// TIA Portal project "TM20T_TiaV151_S71200_V17" (V17)

(* hardware
DEVICE "S7-1200 station_1"  S7-1200 Station
   slot 0: "Rack_0"  S7-1200 Rack  Rack  V1.0
   slot 1: "PLC_1"  CPU 1214C DC/DC/DC  6ES7 214-1AG40-0XB0  V4.2
   slot 2: "DI 8x24VDC_1"  6ES7 221-1BF32-0XB0  V2.0
   slot 3: "DI 16x24VDC_1"  SM 1221 DI16 x 24VDC  6ES7 221-1BH30-0XB0  V1.0
   slot 4: "DI 16x24VDC_2"  SM 1221 DI16 x 24VDC  6ES7 221-1BH30-0XB0  V1.0
   slot 5: "DI 16x24VDC_3"  SM 1221 DI16 x 24VDC  6ES7 221-1BH30-0XB0  V1.0
DEVICE "PC-System_1"  SIMATIC PC station
   slot 0: "SIMATIC PC station"  Rail  SIMATIC PC-Station  V1.0
      slot 125: "Stationmanager"  Station_Manager  V6.0.4
   slot 1: "HMI_RT_1"  WinCC RT Advanced  6AV2 104-0xxxx-xxxx  17.0.0.0
      slot 33792: "Computer interface"  Host interface
   slot 2: "IE general_1"  IE General  IE_CP  V8.2.0
*)

// ===== PLC "PLC_1"  CPU 1214C DC/DC/DC =====

VAR_GLOBAL   // PLC tag table "Default tag table"
   "System_Byte" AT %MB1 : Byte;
   "FirstScan" AT %M1.0 : Bool;
   "DiagStatusUpdate" AT %M1.1 : Bool;
   "AlwaysTRUE" AT %M1.2 : Bool;
   "AlwaysFALSE" AT %M1.3 : Bool;
   "Clock_Byte" AT %MB0 : Byte;
   "Clock_10Hz" AT %M0.0 : Bool;
   "Clock_5Hz" AT %M0.1 : Bool;
   "Clock_2.5Hz" AT %M0.2 : Bool;
   "Clock_2Hz" AT %M0.3 : Bool;
   "Clock_1.25Hz" AT %M0.4 : Bool;
   "Clock_1Hz" AT %M0.5 : Bool;
   "Clock_0.625Hz" AT %M0.6 : Bool;
   "Clock_0.5Hz" AT %M0.7 : Bool;
END_VAR

VAR_GLOBAL   // PLC tag table "INPUT"
   "I_F1_Up" AT %I0.0 : Bool;   // Tầng 1 gọi đi lên
   "I_F2_Up" AT %I0.1 : Bool;   // Tầng 2 gọi đi lên
   "I_F3_Up" AT %I0.2 : Bool;   // Tầng 3 gọi đi lên
   "I_F2_Down" AT %I0.3 : Bool;   // Tầng 2 gọi đi xuống
   "I_F3_Down" AT %I0.4 : Bool;   // Tầng 3 gọi đi xuống
   "I_F4_Down" AT %I0.5 : Bool;   // Tầng 4 gọi đi xuống
   "I_Inside_F1" AT %I0.6 : Bool;   // Gọi tầng trong thang máy gọi tầng 1
   "I_Inside_F2" AT %I0.7 : Bool;   // Gọi tầng trong thang máy gọi tầng 2
   "I_Inside_F3" AT %I1.0 : Bool;   // Gọi tầng trong thang máy gọi tầng 3
   "I_Inside_F4" AT %I1.1 : Bool;   // Gọi tầng trong thang máy gọi tầng 4
   "I_Inside_Door_Open" AT %I1.2 : Bool;   // Nút nhấn mở cửa trong thang máy
   "I_Inside_Door_Close" AT %I1.3 : Bool;   // Nút nhấn đóng cửa trong thang máy
   "I_Cabin_Position" AT %I1.4 : Bool;   // Cảm biến vị trí buồng thang
   "I_Door_Opened" AT %I1.5 : Bool;   // Limits Switch cữa đã mở
   "I_Door_Closed" AT %I1.6 : Bool;   // Limit Switch cửa đã đóng
   "I_F4_Up" AT %I1.7 : Bool;
   "I_F5_Up" AT %I2.0 : Bool;
   "I_F6_Up" AT %I2.1 : Bool;
   "I_F7_Up" AT %I2.2 : Bool;
   "I_F8_Up" AT %I2.3 : Bool;
   "I_F9_Up" AT %I2.4 : Bool;
   "I_F10_Up" AT %I2.5 : Bool;
   "I_F11_Up" AT %I2.6 : Bool;
   "I_F12_Up" AT %I2.7 : Bool;
   "I_F13_Up" AT %I3.0 : Bool;
   "I_F14_Up" AT %I3.1 : Bool;
   "I_F15_Up" AT %I3.2 : Bool;
   "I_F16_Up" AT %I3.3 : Bool;
   "I_F17_Up" AT %I3.4 : Bool;
   "I_F18_Up" AT %I3.5 : Bool;
   "I_F19_Up" AT %I3.6 : Bool;
   "I_F5_Down" AT %I3.7 : Bool;
   "I_F6_Down" AT %I4.0 : Bool;
   "I_F7_Down" AT %I4.1 : Bool;
   "I_F8_Down" AT %I4.2 : Bool;
   "I_F9_Down" AT %I4.3 : Bool;
   "I_F10_Down" AT %I4.4 : Bool;
   "I_F11_Down" AT %I4.5 : Bool;
   "I_F12_Down" AT %I4.6 : Bool;
   "I_F13_Down" AT %I4.7 : Bool;
   "I_F14_Down" AT %I5.0 : Bool;
   "I_F15_Down" AT %I5.1 : Bool;
   "I_F16_Down" AT %I5.2 : Bool;
   "I_F17_Down" AT %I5.3 : Bool;
   "I_F18_Down" AT %I5.4 : Bool;
   "I_F19_Down" AT %I5.5 : Bool;
   "I_F20_Down" AT %I5.6 : Bool;
   "I_Inside_F1(1)" AT %I5.7 : Bool;
   "I_Inside_F2(1)" AT %I6.0 : Bool;
   "I_Inside_F3(1)" AT %I6.1 : Bool;
   "I_Inside_F4(1)" AT %I6.2 : Bool;
   "I_Inside_F5" AT %I6.3 : Bool;
   "I_Inside_F6" AT %I6.4 : Bool;
   "I_Inside_F7" AT %I6.5 : Bool;
   "I_Inside_F8" AT %I6.6 : Bool;
   "I_Inside_F9" AT %I6.7 : Bool;
   "I_Inside_F10" AT %I7.0 : Bool;
   "I_Inside_F11" AT %I7.1 : Bool;
   "I_Inside_F12" AT %I7.2 : Bool;
   "I_Inside_F13" AT %I7.3 : Bool;
   "I_Inside_F14" AT %I7.4 : Bool;
   "I_Inside_F15" AT %I7.5 : Bool;
   "I_Inside_F16" AT %I7.6 : Bool;
   "I_Inside_F17" AT %I7.7 : Bool;
   "I_Inside_F18" AT %I8.0 : Bool;
   "I_Inside_F19" AT %I8.1 : Bool;
   "I_Inside_F20" AT %I8.2 : Bool;
END_VAR

VAR_GLOBAL   // PLC tag table "OUTPUT"
   "Q_Door_Open" AT %Q0.0 : Bool;   // Cửa buồng thang mở
   "Q_Door_Close" AT %Q0.1 : Bool;   // Cửa buồng thang đóng
   "Q_Eleveytor_Up" AT %Q0.2 : Bool;   // Thang máy đi lên
   "Q_Eleveytor_Down" AT %Q0.3 : Bool;   // Thang máy đi xuống
END_VAR

VAR_GLOBAL   // PLC tag table "xung suon len"
   "P1" AT %M20.0 : Bool;
   "P2" AT %M20.1 : Bool;
   "P3" AT %M20.2 : Bool;
   "P4" AT %M20.3 : Bool;
   "P5" AT %M20.4 : Bool;
   "P6" AT %M20.5 : Bool;
   "P7" AT %M20.6 : Bool;
   "P8" AT %M20.7 : Bool;
   "P9" AT %M21.0 : Bool;
   "P10" AT %M21.1 : Bool;
   "P11" AT %M21.2 : Bool;
   "P12" AT %M21.3 : Bool;
   "P13" AT %M21.4 : Bool;
   "P14" AT %M21.5 : Bool;
   "P15" AT %M21.6 : Bool;
   "P16" AT %M21.7 : Bool;
   "P17" AT %M22.0 : Bool;
   "P18" AT %M22.1 : Bool;
   "P19" AT %M22.2 : Bool;
   "P20" AT %M22.3 : Bool;
   "P21" AT %M22.4 : Bool;
   "P22" AT %M22.5 : Bool;
   "P23" AT %M22.6 : Bool;
   "P24" AT %M22.7 : Bool;
   "P25" AT %M23.0 : Bool;
   "P26" AT %M23.1 : Bool;
   "P27" AT %M23.2 : Bool;
   "P28" AT %M23.3 : Bool;
   "P29" AT %M23.4 : Bool;
   "P30" AT %M23.5 : Bool;
   "P31" AT %M23.6 : Bool;
   "P32" AT %M23.7 : Bool;
   "P33" AT %M24.0 : Bool;
   "P34" AT %M24.1 : Bool;
   "P35" AT %M24.2 : Bool;
   "P36" AT %M24.3 : Bool;
   "P37" AT %M24.4 : Bool;
   "P38" AT %M24.5 : Bool;
   "P39" AT %M24.6 : Bool;
   "P40" AT %M24.7 : Bool;
   "P41" AT %M25.0 : Bool;
   "P42" AT %M25.1 : Bool;
   "P43" AT %M25.2 : Bool;
   "P44" AT %M25.3 : Bool;
   "P45" AT %M25.4 : Bool;
   "P46" AT %M25.5 : Bool;
   "P47" AT %M25.6 : Bool;
   "P48" AT %M25.7 : Bool;
   "P49" AT %M26.0 : Bool;
   "P50" AT %M26.1 : Bool;
   "P51" AT %M26.2 : Bool;
   "P52" AT %M26.3 : Bool;
   "P53" AT %M26.4 : Bool;
   "P54" AT %M26.5 : Bool;
   "P55" AT %M26.6 : Bool;
   "P56" AT %M26.7 : Bool;
   "P57" AT %M27.0 : Bool;
   "P58" AT %M27.1 : Bool;
   "P59" AT %M27.2 : Bool;
   "P60" AT %M27.3 : Bool;
   "P61" AT %M27.4 : Bool;
   "P62" AT %M27.5 : Bool;
   "P63" AT %M27.6 : Bool;
   "P64" AT %M27.7 : Bool;
   "P65" AT %M28.0 : Bool;
   "P66" AT %M28.1 : Bool;
   "P67" AT %M28.2 : Bool;
   "P68" AT %M28.3 : Bool;
   "P69" AT %M28.4 : Bool;
   "P70" AT %M28.5 : Bool;
   "P71" AT %M28.6 : Bool;
   "P72" AT %M28.7 : Bool;
   "P73" AT %M29.0 : Bool;
   "P74" AT %M29.1 : Bool;
   "P75" AT %M29.2 : Bool;
   "P76" AT %M29.3 : Bool;
   "P77" AT %M29.4 : Bool;
   "P78" AT %M29.5 : Bool;
   "P79" AT %M29.6 : Bool;
   "P80" AT %M29.7 : Bool;
   "P81" AT %M30.0 : Bool;
   "P82" AT %M30.1 : Bool;
   "P83" AT %M30.2 : Bool;
   "P84" AT %M30.3 : Bool;
   "P85" AT %M30.4 : Bool;
   "P86" AT %M30.5 : Bool;
   "P87" AT %M30.6 : Bool;
   "P88" AT %M30.7 : Bool;
   "P89" AT %M31.0 : Bool;
   "P90" AT %M31.1 : Bool;
   "P91" AT %M31.2 : Bool;
   "P92" AT %M31.3 : Bool;
   "P93" AT %M31.4 : Bool;
   "P94" AT %M31.5 : Bool;
   "P95" AT %M31.6 : Bool;
   "P96" AT %M31.7 : Bool;
   "P97" AT %M32.0 : Bool;
   "P98" AT %M32.1 : Bool;
   "P99" AT %M32.2 : Bool;
   "P100" AT %M32.3 : Bool;
   "P101" AT %M32.4 : Bool;
   "P102" AT %M32.5 : Bool;
   "P103" AT %M32.6 : Bool;
   "P104" AT %M32.7 : Bool;
   "P105" AT %M33.0 : Bool;
   "P106" AT %M33.1 : Bool;
   "P107" AT %M33.2 : Bool;
   "P108" AT %M33.3 : Bool;
   "P109" AT %M33.4 : Bool;
   "P110" AT %M33.5 : Bool;
   "P111" AT %M33.6 : Bool;
   "P112" AT %M33.7 : Bool;
   "P113" AT %M34.0 : Bool;
   "P114" AT %M34.1 : Bool;
   "P115" AT %M34.2 : Bool;
   "P116" AT %M34.3 : Bool;
   "P117" AT %M34.4 : Bool;
   "P118" AT %M34.5 : Bool;
   "P119" AT %M34.6 : Bool;
   "P120" AT %M34.7 : Bool;
   "P121" AT %M35.0 : Bool;
   "P122" AT %M35.1 : Bool;
   "P123" AT %M35.2 : Bool;
   "P124" AT %M35.3 : Bool;
   "P125" AT %M35.4 : Bool;
   "P126" AT %M35.5 : Bool;
   "P127" AT %M35.6 : Bool;
   "P128" AT %M35.7 : Bool;
   "P129" AT %M36.0 : Bool;
   "P130" AT %M36.1 : Bool;
   "P131" AT %M36.2 : Bool;
   "P132" AT %M36.3 : Bool;
   "P133" AT %M36.4 : Bool;
   "P134" AT %M36.5 : Bool;
   "P135" AT %M36.6 : Bool;
   "P136" AT %M36.7 : Bool;
   "P137" AT %M37.0 : Bool;
   "P138" AT %M37.1 : Bool;
   "P139" AT %M37.2 : Bool;
   "P140" AT %M37.3 : Bool;
   "P141" AT %M37.4 : Bool;
   "P142" AT %M37.5 : Bool;
   "P143" AT %M37.6 : Bool;
   "P144" AT %M37.7 : Bool;
   "P145" AT %M38.0 : Bool;
   "P146" AT %M38.1 : Bool;
   "P147" AT %M38.2 : Bool;
   "P148" AT %M38.3 : Bool;
   "P149" AT %M38.4 : Bool;
   "P150" AT %M38.5 : Bool;
   "P151" AT %M38.6 : Bool;
   "P152" AT %M38.7 : Bool;
   "P153" AT %M39.0 : Bool;
   "P154" AT %M39.1 : Bool;
   "P155" AT %M39.2 : Bool;
   "P156" AT %M39.3 : Bool;
   "P157" AT %M39.4 : Bool;
   "P158" AT %M39.5 : Bool;
   "P159" AT %M39.6 : Bool;
   "P160" AT %M39.7 : Bool;
   "P161" AT %M40.0 : Bool;
   "P162" AT %M40.1 : Bool;
   "P163" AT %M40.2 : Bool;
   "P164" AT %M40.3 : Bool;
   "P165" AT %M40.4 : Bool;
   "P166" AT %M40.5 : Bool;
   "P167" AT %M40.6 : Bool;
   "P168" AT %M40.7 : Bool;
   "P169" AT %M41.0 : Bool;
   "P170" AT %M41.1 : Bool;
   "P171" AT %M41.2 : Bool;
   "P172" AT %M41.3 : Bool;
   "P173" AT %M41.4 : Bool;
   "P174" AT %M41.5 : Bool;
   "P175" AT %M41.6 : Bool;
   "P176" AT %M41.7 : Bool;
   "P177" AT %M42.0 : Bool;
   "P178" AT %M42.1 : Bool;
   "P179" AT %M42.2 : Bool;
   "P180" AT %M42.3 : Bool;
   "P181" AT %M42.4 : Bool;
   "P182" AT %M42.5 : Bool;
   "P183" AT %M42.6 : Bool;
   "P184" AT %M42.7 : Bool;
   "P185" AT %M43.0 : Bool;
   "P186" AT %M43.1 : Bool;
   "P187" AT %M43.2 : Bool;
   "P188" AT %M43.3 : Bool;
   "P189" AT %M43.4 : Bool;
   "P190" AT %M43.5 : Bool;
   "P191" AT %M43.6 : Bool;
   "P192" AT %M43.7 : Bool;
   "P193" AT %M44.0 : Bool;
   "P194" AT %M44.1 : Bool;
   "P195" AT %M44.2 : Bool;
   "P196" AT %M44.3 : Bool;
   "P197" AT %M44.4 : Bool;
   "P198" AT %M44.5 : Bool;
   "P199" AT %M44.6 : Bool;
   "P200" AT %M44.7 : Bool;
   "P201" AT %M45.0 : Bool;
   "P202" AT %M45.1 : Bool;
   "P203" AT %M45.2 : Bool;
   "P204" AT %M45.3 : Bool;
   "P205" AT %M45.4 : Bool;
   "P206" AT %M45.5 : Bool;
   "P207" AT %M45.6 : Bool;
   "P208" AT %M45.7 : Bool;
   "P209" AT %M46.0 : Bool;
   "P210" AT %M46.1 : Bool;
   "P211" AT %M46.2 : Bool;
   "P212" AT %M46.3 : Bool;
   "P213" AT %M46.4 : Bool;
   "P214" AT %M46.5 : Bool;
   "P215" AT %M46.6 : Bool;
   "P216" AT %M46.7 : Bool;
   "P217" AT %M47.0 : Bool;
   "P218" AT %M47.1 : Bool;
   "P219" AT %M47.2 : Bool;
END_VAR

VAR_GLOBAL   // PLC tag table "Simulation"
   "Simu_Eleveytor" AT %MW100 : Int;
   "Simu_Door_F1" AT %MW102 : Int;
   "Simu_Door_F2" AT %MW104 : Int;
   "Simu_Door_F3" AT %MW106 : Int;
   "Simu_Door_F4" AT %MW108 : Int;
   "M_Simulation" AT %M10.0 : Bool;
   "Display_Inside_F2" AT %M10.1 : Bool;   // Hiển thị màu nút nhấn trong buồng thang tầng 2
   "Display_Inside_F3" AT %M10.2 : Bool;   // Hiển thị màu nút nhấn trong buồng thang tầng 3
   "Simu_Door_F5" AT %MW110 : Int;
   "Simu_Door_F6" AT %MW112 : Int;
   "Simu_Door_F7" AT %MW114 : Int;
   "Simu_Door_F8" AT %MW116 : Int;
   "Simu_Door_F9" AT %MW118 : Int;
   "Simu_Door_F10" AT %MW120 : Int;
   "Simu_Door_F11" AT %MW122 : Int;
   "Simu_Door_F12" AT %MW124 : Int;
   "Simu_Door_F13" AT %MW126 : Int;
   "Simu_Door_F14" AT %MW128 : Int;
   "Simu_Door_F15" AT %MW130 : Int;
   "Simu_Door_F16" AT %MW132 : Int;
   "Simu_Door_F17" AT %MW134 : Int;
   "Simu_Door_F18" AT %MW136 : Int;
   "Simu_Door_F19" AT %MW138 : Int;
   "Simu_Door_F20" AT %MW140 : Int;
   "Display_Inside_F4" AT %M10.3 : Bool;
   "Display_Inside_F5" AT %M10.4 : Bool;
   "Display_Inside_F6" AT %M10.5 : Bool;
   "Display_Inside_F7" AT %M10.6 : Bool;
   "Display_Inside_F8" AT %M10.7 : Bool;
   "Display_Inside_F9" AT %M11.0 : Bool;
   "Display_Inside_F10" AT %M11.1 : Bool;
   "Display_Inside_F11" AT %M11.2 : Bool;
   "Display_Inside_F12" AT %M11.3 : Bool;
   "Display_Inside_F13" AT %M11.4 : Bool;
   "Display_Inside_F14" AT %M11.5 : Bool;
   "Display_Inside_F15" AT %M11.6 : Bool;
   "Display_Inside_F16" AT %M11.7 : Bool;
   "Display_Inside_F17" AT %M12.0 : Bool;
   "Display_Inside_F18" AT %M12.1 : Bool;
   "Display_Inside_F19" AT %M12.2 : Bool;
   "M_Check1" AT %M12.3 : Bool;
   "M_Check2" AT %M12.4 : Bool;
END_VAR

TYPE "Thang_May"
   STRUCT
      Position : Bool;   // Vị trí thang máy ở tầng hiện tại
      Btt_Up_Selected : Bool;   // Đã chọn đi lên
      Btt_Down_Selected : Bool;   // Đã chọn đi xuống
      TG_Up_Selected : Bool;   // Lựa chọn đi lên đã chọn
      TG_Down_Selected : Bool;   // Lựa chọn đi xuống đã chọn
      Sensor_Correct_Position : Bool;   // Vị trí chính xác để mở cửa
      Door_Opened : Bool;   // Cửa đã mở
      Door_Closed : Bool;   // Cửa đã đóng
      I_Button_Up : Bool;   // Nút nhấn đi lên
      I_Button_Down : Bool;   // Nút nhấn đi xuống
   END_STRUCT;
END_TYPE

DATA_BLOCK "DB_Data"   // DB1
{ S7_Optimized_Access := 'TRUE' }
VERSION : 0.1
   VAR
      F1 : "Thang_May";
      F2 : "Thang_May";
      F3 : "Thang_May";
      F4 : "Thang_May";
      F20 : "Thang_May";
      F19 : "Thang_May";
      F18 : "Thang_May";
      F17 : "Thang_May";
      F16 : "Thang_May";
      F15 : "Thang_May";
      F14 : "Thang_May";
      F13 : "Thang_May";
      F12 : "Thang_May";
      F11 : "Thang_May";
      F10 : "Thang_May";
      F9 : "Thang_May";
      F8 : "Thang_May";
      F7 : "Thang_May";
      F6 : "Thang_May";
      F5 : "Thang_May";
      Button_Inside_F1 : Bool;
      Button_Inside_F2 : Bool;
      Button_Inside_F3 : Bool;
      Button_Inside_F20 : Bool;
      Button_Inside_F19 : Bool;
      Button_Inside_F18 : Bool;
      Button_Inside_F17 : Bool;
      Button_Inside_F16 : Bool;
      Button_Inside_F15 : Bool;
      Button_Inside_F14 : Bool;
      Button_Inside_F13 : Bool;
      Button_Inside_F12 : Bool;
      Button_Inside_F11 : Bool;
      Button_Inside_F10 : Bool;
      Button_Inside_F9 : Bool;
      Button_Inside_F8 : Bool;
      Button_Inside_F7 : Bool;
      Button_Inside_F6 : Bool;
      Button_Inside_F5 : Bool;
      Button_Inside_F4 : Bool;
      Button_Inside_Open : Bool;
      Button_Inside_Close : Bool;
      LS_Door_Opened : Bool;
      LS_Door_Closed : Bool;
      Eleveytor_Upping : Bool;
      Eleveytor_Downing : Bool;
      Last_Is_Up : Bool;   // Trước đó thang máy đang đi lên
      Last_Is_Down : Bool;   // Trước đó thang máy đang đi xuống
   END_VAR
BEGIN
END_DATA_BLOCK

// folder: System blocks/Program resources

DATA_BLOCK "IEC_Timer_0_DB"   // DB2
{ S7_Optimized_Access := 'TRUE' }
AUTHOR : Simatic
FAMILY : IEC
NAME : IEC_TMR
VERSION : 1.0
// stored: InstanceOfName IEC_TIMER
"IEC_TIMER"
BEGIN
END_DATA_BLOCK

DATA_BLOCK "IEC_Timer_0_DB_1"   // DB3
{ S7_Optimized_Access := 'TRUE' }
AUTHOR : Simatic
FAMILY : IEC
NAME : IEC_TMR
VERSION : 1.0
// stored: InstanceOfName IEC_TIMER
"IEC_TIMER"
BEGIN
END_DATA_BLOCK

DATA_BLOCK "IEC_Timer_0_DB_2"   // DB4
{ S7_Optimized_Access := 'TRUE' }
AUTHOR : Simatic
FAMILY : IEC
NAME : IEC_TMR
VERSION : 1.0
// stored: InstanceOfName IEC_TIMER
"IEC_TIMER"
BEGIN
END_DATA_BLOCK

DATA_BLOCK "IEC_Timer_0_DB_3"   // DB5
{ S7_Optimized_Access := 'TRUE' }
AUTHOR : Simatic
FAMILY : IEC
NAME : IEC_TMR
VERSION : 1.0
// stored: InstanceOfName IEC_TIMER
"IEC_TIMER"
BEGIN
END_DATA_BLOCK

DATA_BLOCK "IEC_Timer_0_DB_4"   // DB6
{ S7_Optimized_Access := 'TRUE' }
AUTHOR : Simatic
FAMILY : IEC
NAME : IEC_TMR
VERSION : 1.0
// stored: InstanceOfName IEC_TIMER
"IEC_TIMER"
BEGIN
END_DATA_BLOCK

// folder: (top level)

FUNCTION "FC_Nut_Nhan" : Void   // FC1, LAD
{ S7_Optimized_Access := 'TRUE' }
VERSION : 0.1
   VAR_TEMP   // added for the SCL form of the ladder/FBD networks
      _w1 : Bool;
      _w2 : Bool;
      _w3 : Bool;
      _w4 : Bool;
      _w5 : Bool;
      _w6 : Bool;
      _w7 : Bool;
      _w8 : Bool;
      _w9 : Bool;
      _w10 : Bool;
      _w11 : Bool;
      _w12 : Bool;
      _w13 : Bool;
      _w14 : Bool;
      _w15 : Bool;
      _w16 : Bool;
      _w17 : Bool;
      _w18 : Bool;
      _w19 : Bool;
      _w20 : Bool;
      _w21 : Bool;
      _w22 : Bool;
      _w23 : Bool;
      _w24 : Bool;
      _w25 : Bool;
      _w26 : Bool;
      _w27 : Bool;
   END_VAR
BEGIN

REGION Network 1: Nút nhấn MỞ cửa tại các tầng
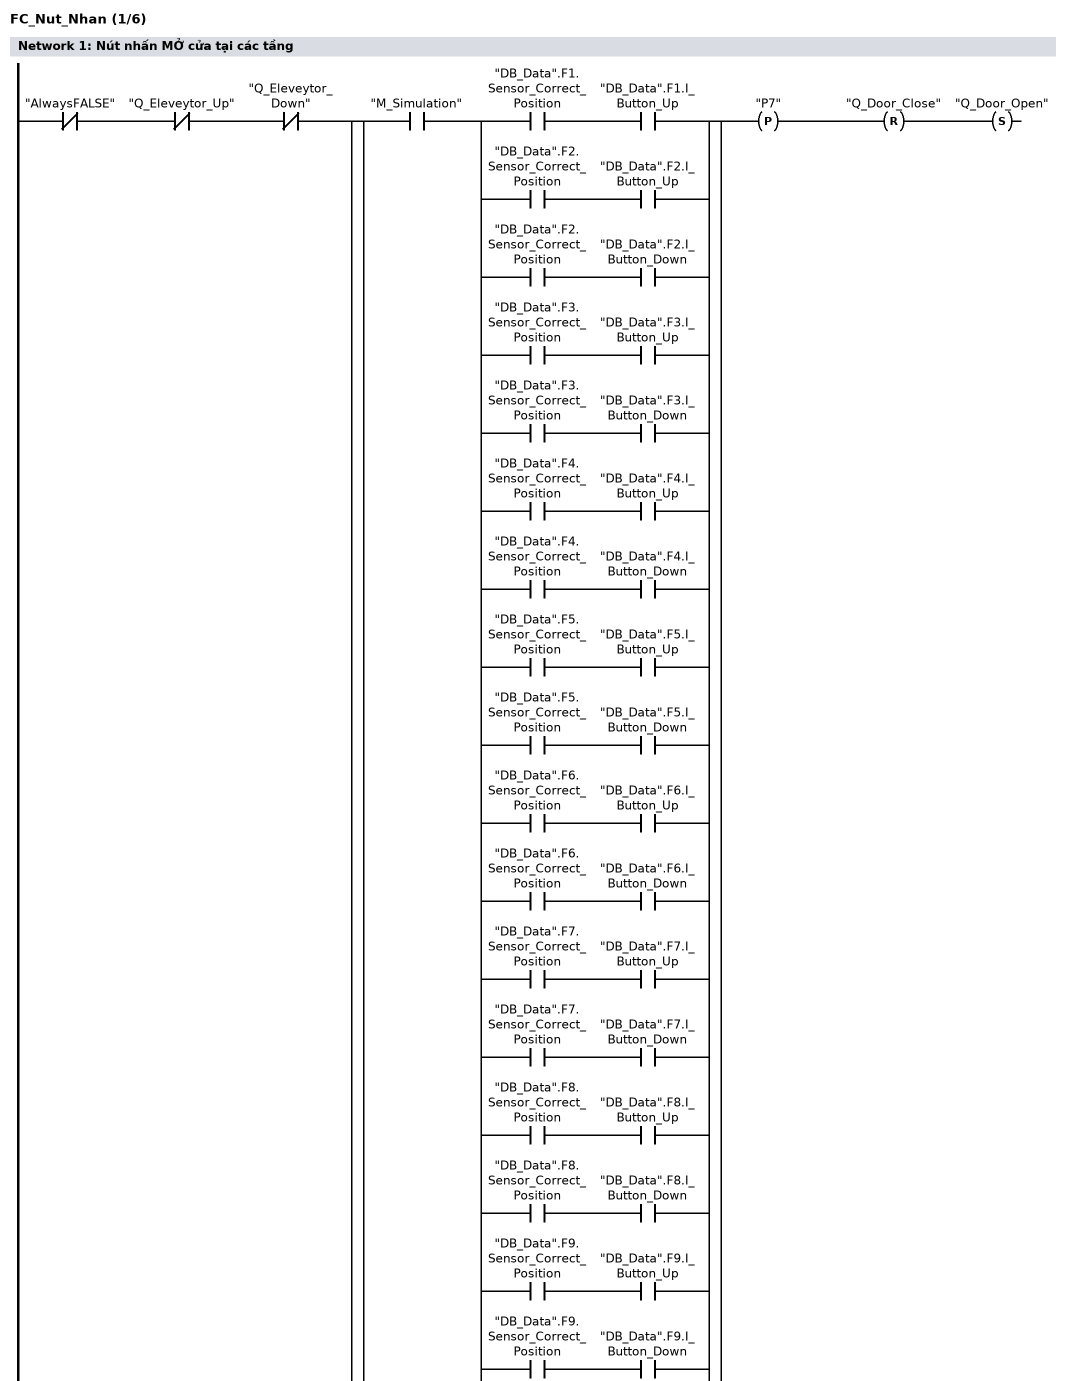
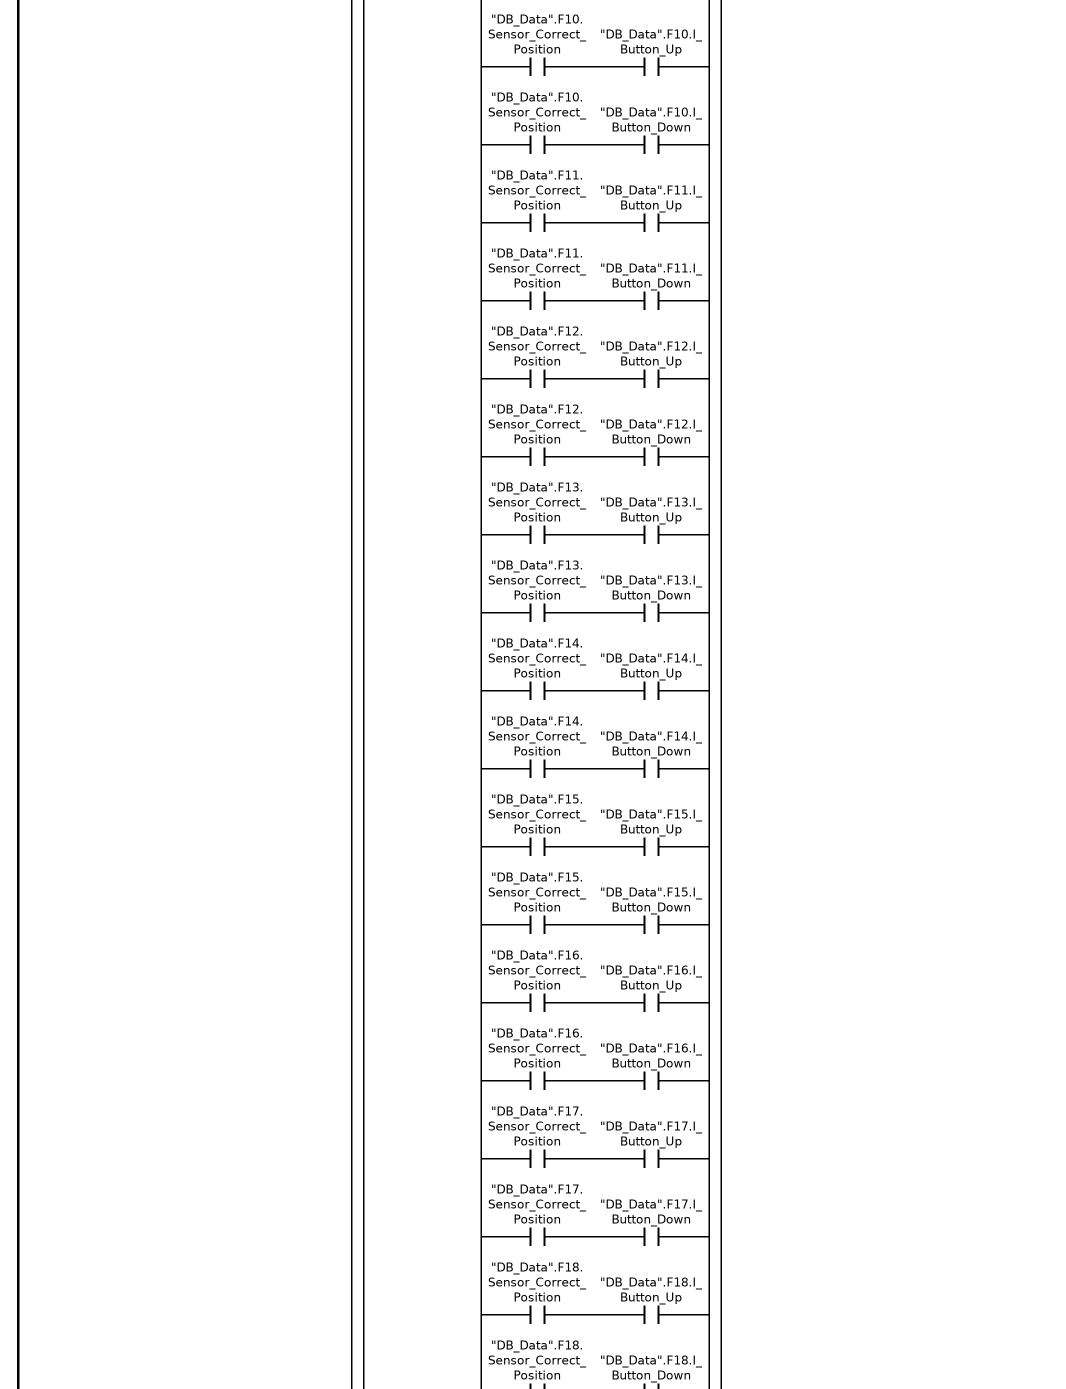
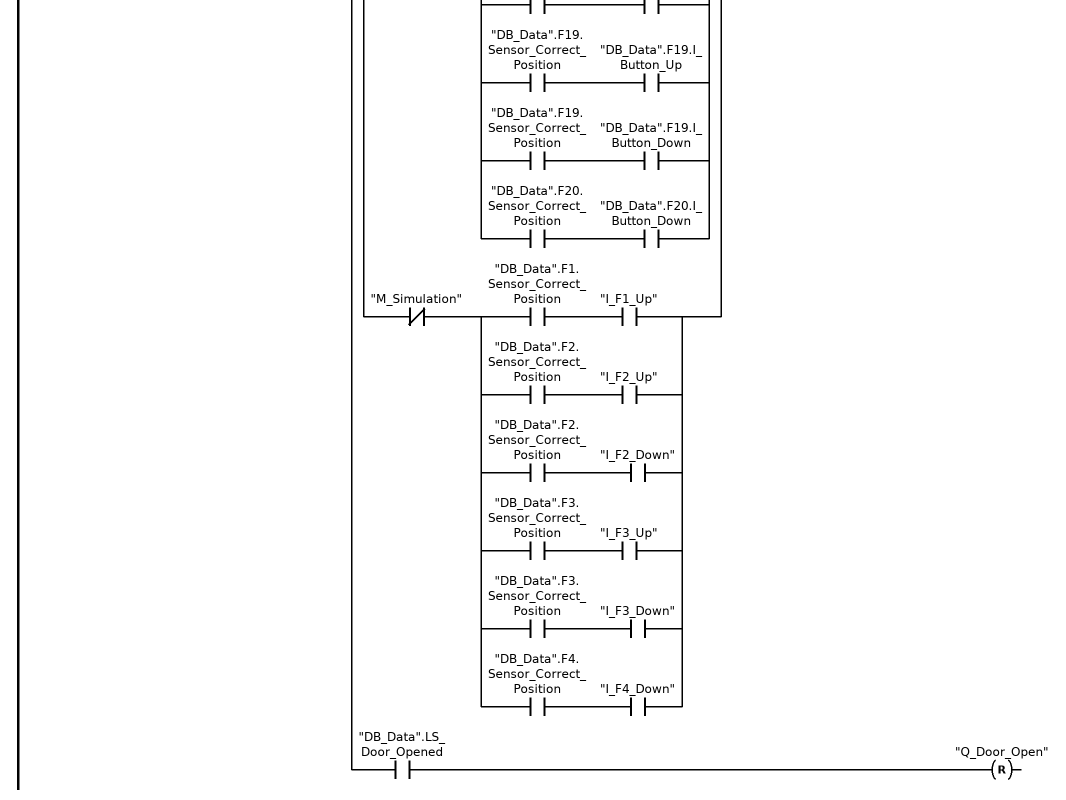
   RUNG wire#powerrail
      I_Contact( "AlwaysFALSE" )
      I_Contact( "Q_Eleveytor_Up" )
      I_Contact( "Q_Eleveytor_Down" )
      wire#w1
      Contact( "M_Simulation" )
      wire#w2
      Contact( "DB_Data".F1.Sensor_Correct_Position )
      Contact( "DB_Data".F1.I_Button_Up )
      wire#w3
      P_Trig( "P7" )
      R_Coil( "Q_Door_Close" )
      S_Coil( "Q_Door_Open" )
   END_RUNG
   RUNG wire#w2
      Contact( "DB_Data".F2.Sensor_Correct_Position )
      Contact( "DB_Data".F2.I_Button_Up )
   END_RUNG wire#w3
   RUNG wire#w2
      Contact( "DB_Data".F2.Sensor_Correct_Position )
      Contact( "DB_Data".F2.I_Button_Down )
   END_RUNG wire#w3
   RUNG wire#w2
      Contact( "DB_Data".F3.Sensor_Correct_Position )
      Contact( "DB_Data".F3.I_Button_Up )
   END_RUNG wire#w3
   RUNG wire#w2
      Contact( "DB_Data".F3.Sensor_Correct_Position )
      Contact( "DB_Data".F3.I_Button_Down )
   END_RUNG wire#w3
   RUNG wire#w2
      Contact( "DB_Data".F4.Sensor_Correct_Position )
      Contact( "DB_Data".F4.I_Button_Up )
   END_RUNG wire#w3
   RUNG wire#w2
      Contact( "DB_Data".F4.Sensor_Correct_Position )
      Contact( "DB_Data".F4.I_Button_Down )
   END_RUNG wire#w3
   RUNG wire#w2
      Contact( "DB_Data".F5.Sensor_Correct_Position )
      Contact( "DB_Data".F5.I_Button_Up )
   END_RUNG wire#w3
   RUNG wire#w2
      Contact( "DB_Data".F5.Sensor_Correct_Position )
      Contact( "DB_Data".F5.I_Button_Down )
   END_RUNG wire#w3
   RUNG wire#w2
      Contact( "DB_Data".F6.Sensor_Correct_Position )
      Contact( "DB_Data".F6.I_Button_Up )
   END_RUNG wire#w3
   RUNG wire#w2
      Contact( "DB_Data".F6.Sensor_Correct_Position )
      Contact( "DB_Data".F6.I_Button_Down )
   END_RUNG wire#w3
   RUNG wire#w2
      Contact( "DB_Data".F7.Sensor_Correct_Position )
      Contact( "DB_Data".F7.I_Button_Up )
   END_RUNG wire#w3
   RUNG wire#w2
      Contact( "DB_Data".F7.Sensor_Correct_Position )
      Contact( "DB_Data".F7.I_Button_Down )
   END_RUNG wire#w3
   RUNG wire#w2
      Contact( "DB_Data".F8.Sensor_Correct_Position )
      Contact( "DB_Data".F8.I_Button_Up )
   END_RUNG wire#w3
   RUNG wire#w2
      Contact( "DB_Data".F8.Sensor_Correct_Position )
      Contact( "DB_Data".F8.I_Button_Down )
   END_RUNG wire#w3
   RUNG wire#w2
      Contact( "DB_Data".F9.Sensor_Correct_Position )
      Contact( "DB_Data".F9.I_Button_Up )
   END_RUNG wire#w3
   RUNG wire#w2
      Contact( "DB_Data".F9.Sensor_Correct_Position )
      Contact( "DB_Data".F9.I_Button_Down )
   END_RUNG wire#w3
   RUNG wire#w2
      Contact( "DB_Data".F10.Sensor_Correct_Position )
      Contact( "DB_Data".F10.I_Button_Up )
   END_RUNG wire#w3
   RUNG wire#w2
      Contact( "DB_Data".F10.Sensor_Correct_Position )
      Contact( "DB_Data".F10.I_Button_Down )
   END_RUNG wire#w3
   RUNG wire#w2
      Contact( "DB_Data".F11.Sensor_Correct_Position )
      Contact( "DB_Data".F11.I_Button_Up )
   END_RUNG wire#w3
   RUNG wire#w2
      Contact( "DB_Data".F11.Sensor_Correct_Position )
      Contact( "DB_Data".F11.I_Button_Down )
   END_RUNG wire#w3
   RUNG wire#w2
      Contact( "DB_Data".F12.Sensor_Correct_Position )
      Contact( "DB_Data".F12.I_Button_Up )
   END_RUNG wire#w3
   RUNG wire#w2
      Contact( "DB_Data".F12.Sensor_Correct_Position )
      Contact( "DB_Data".F12.I_Button_Down )
   END_RUNG wire#w3
   RUNG wire#w2
      Contact( "DB_Data".F13.Sensor_Correct_Position )
      Contact( "DB_Data".F13.I_Button_Up )
   END_RUNG wire#w3
   RUNG wire#w2
      Contact( "DB_Data".F13.Sensor_Correct_Position )
      Contact( "DB_Data".F13.I_Button_Down )
   END_RUNG wire#w3
   RUNG wire#w2
      Contact( "DB_Data".F14.Sensor_Correct_Position )
      Contact( "DB_Data".F14.I_Button_Up )
   END_RUNG wire#w3
   RUNG wire#w2
      Contact( "DB_Data".F14.Sensor_Correct_Position )
      Contact( "DB_Data".F14.I_Button_Down )
   END_RUNG wire#w3
   RUNG wire#w2
      Contact( "DB_Data".F15.Sensor_Correct_Position )
      Contact( "DB_Data".F15.I_Button_Up )
   END_RUNG wire#w3
   RUNG wire#w2
      Contact( "DB_Data".F15.Sensor_Correct_Position )
      Contact( "DB_Data".F15.I_Button_Down )
   END_RUNG wire#w3
   RUNG wire#w2
      Contact( "DB_Data".F16.Sensor_Correct_Position )
      Contact( "DB_Data".F16.I_Button_Up )
   END_RUNG wire#w3
   RUNG wire#w2
      Contact( "DB_Data".F16.Sensor_Correct_Position )
      Contact( "DB_Data".F16.I_Button_Down )
   END_RUNG wire#w3
   RUNG wire#w2
      Contact( "DB_Data".F17.Sensor_Correct_Position )
      Contact( "DB_Data".F17.I_Button_Up )
   END_RUNG wire#w3
   RUNG wire#w2
      Contact( "DB_Data".F17.Sensor_Correct_Position )
      Contact( "DB_Data".F17.I_Button_Down )
   END_RUNG wire#w3
   RUNG wire#w2
      Contact( "DB_Data".F18.Sensor_Correct_Position )
      Contact( "DB_Data".F18.I_Button_Up )
   END_RUNG wire#w3
   RUNG wire#w2
      Contact( "DB_Data".F18.Sensor_Correct_Position )
      Contact( "DB_Data".F18.I_Button_Down )
   END_RUNG wire#w3
   RUNG wire#w2
      Contact( "DB_Data".F19.Sensor_Correct_Position )
      Contact( "DB_Data".F19.I_Button_Up )
   END_RUNG wire#w3
   RUNG wire#w2
      Contact( "DB_Data".F19.Sensor_Correct_Position )
      Contact( "DB_Data".F19.I_Button_Down )
   END_RUNG wire#w3
   RUNG wire#w2
      Contact( "DB_Data".F20.Sensor_Correct_Position )
      Contact( "DB_Data".F20.I_Button_Down )
   END_RUNG wire#w3
   RUNG wire#w1
      I_Contact( "M_Simulation" )
      wire#w4
      Contact( "DB_Data".F1.Sensor_Correct_Position )
      Contact( "I_F1_Up" )
   END_RUNG wire#w3
   RUNG wire#w4
      Contact( "DB_Data".F2.Sensor_Correct_Position )
      Contact( "I_F2_Up" )
   END_RUNG wire#w3
   RUNG wire#w4
      Contact( "DB_Data".F2.Sensor_Correct_Position )
      Contact( "I_F2_Down" )
   END_RUNG wire#w3
   RUNG wire#w4
      Contact( "DB_Data".F3.Sensor_Correct_Position )
      Contact( "I_F3_Up" )
   END_RUNG wire#w3
   RUNG wire#w4
      Contact( "DB_Data".F3.Sensor_Correct_Position )
      Contact( "I_F3_Down" )
   END_RUNG wire#w3
   RUNG wire#w4
      Contact( "DB_Data".F4.Sensor_Correct_Position )
      Contact( "I_F4_Down" )
   END_RUNG wire#w3
   RUNG wire#w1
      Contact( "DB_Data".LS_Door_Opened )
      R_Coil( "Q_Door_Open" )
   END_RUNG
   // the same network as SCL:
   #_w1 := NOT "AlwaysFALSE" AND NOT "Q_Eleveytor_Up" AND NOT "Q_Eleveytor_Down";
   #_w2 := #_w1 AND (("M_Simulation" AND (("DB_Data".F1.Sensor_Correct_Position AND "DB_Data".F1.I_Button_Up) OR ("DB_Data".F2.Sensor_Correct_Position AND "DB_Data".F2.I_Button_Up) OR ("DB_Data".F2.Sensor_Correct_Position AND "DB_Data".F2.I_Button_Down) OR ("DB_Data".F3.Sensor_Correct_Position AND "DB_Data".F3.I_Button_Up) OR ("DB_Data".F3.Sensor_Correct_Position AND "DB_Data".F3.I_Button_Down) OR ("DB_Data".F4.Sensor_Correct_Position AND "DB_Data".F4.I_Button_Up) OR ("DB_Data".F4.Sensor_Correct_Position AND "DB_Data".F4.I_Button_Down) OR ("DB_Data".F5.Sensor_Correct_Position AND "DB_Data".F5.I_Button_Up) OR ("DB_Data".F5.Sensor_Correct_Position AND "DB_Data".F5.I_Button_Down) OR ("DB_Data".F6.Sensor_Correct_Position AND "DB_Data".F6.I_Button_Up) OR ("DB_Data".F6.Sensor_Correct_Position AND "DB_Data".F6.I_Button_Down) OR ("DB_Data".F7.Sensor_Correct_Position AND "DB_Data".F7.I_Button_Up) OR ("DB_Data".F7.Sensor_Correct_Position AND "DB_Data".F7.I_Button_Down) OR ("DB_Data".F8.Sensor_Correct_Position AND "DB_Data".F8.I_Button_Up) OR ("DB_Data".F8.Sensor_Correct_Position AND "DB_Data".F8.I_Button_Down) OR ("DB_Data".F9.Sensor_Correct_Position AND "DB_Data".F9.I_Button_Up) OR ("DB_Data".F9.Sensor_Correct_Position AND "DB_Data".F9.I_Button_Down) OR ("DB_Data".F10.Sensor_Correct_Position AND "DB_Data".F10.I_Button_Up) OR ("DB_Data".F10.Sensor_Correct_Position AND "DB_Data".F10.I_Button_Down) OR ("DB_Data".F11.Sensor_Correct_Position AND "DB_Data".F11.I_Button_Up) OR ("DB_Data".F11.Sensor_Correct_Position AND "DB_Data".F11.I_Button_Down) OR ("DB_Data".F12.Sensor_Correct_Position AND "DB_Data".F12.I_Button_Up) OR ("DB_Data".F12.Sensor_Correct_Position AND "DB_Data".F12.I_Button_Down) OR ("DB_Data".F13.Sensor_Correct_Position AND "DB_Data".F13.I_Button_Up) OR ("DB_Data".F13.Sensor_Correct_Position AND "DB_Data".F13.I_Button_Down) OR ("DB_Data".F14.Sensor_Correct_Position AND "DB_Data".F14.I_Button_Up) OR ("DB_Data".F14.Sensor_Correct_Position AND "DB_Data".F14.I_Button_Down) OR ("DB_Data".F15.Sensor_Correct_Position AND "DB_Data".F15.I_Button_Up) OR ("DB_Data".F15.Sensor_Correct_Position AND "DB_Data".F15.I_Button_Down) OR ("DB_Data".F16.Sensor_Correct_Position AND "DB_Data".F16.I_Button_Up) OR ("DB_Data".F16.Sensor_Correct_Position AND "DB_Data".F16.I_Button_Down) OR ("DB_Data".F17.Sensor_Correct_Position AND "DB_Data".F17.I_Button_Up) OR ("DB_Data".F17.Sensor_Correct_Position AND "DB_Data".F17.I_Button_Down) OR ("DB_Data".F18.Sensor_Correct_Position AND "DB_Data".F18.I_Button_Up) OR ("DB_Data".F18.Sensor_Correct_Position AND "DB_Data".F18.I_Button_Down) OR ("DB_Data".F19.Sensor_Correct_Position AND "DB_Data".F19.I_Button_Up) OR ("DB_Data".F19.Sensor_Correct_Position AND "DB_Data".F19.I_Button_Down) OR ("DB_Data".F20.Sensor_Correct_Position AND "DB_Data".F20.I_Button_Down))) OR (NOT "M_Simulation" AND (("DB_Data".F1.Sensor_Correct_Position AND "I_F1_Up") OR ("DB_Data".F2.Sensor_Correct_Position AND "I_F2_Up") OR ("DB_Data".F2.Sensor_Correct_Position AND "I_F2_Down") OR ("DB_Data".F3.Sensor_Correct_Position AND "I_F3_Up") OR ("DB_Data".F3.Sensor_Correct_Position AND "I_F3_Down") OR ("DB_Data".F4.Sensor_Correct_Position AND "I_F4_Down"))));
   #_w3 := #_w2 AND NOT "P7";   // rising edge
   "P7" := #_w2;
   IF #_w3 THEN
       "Q_Door_Close" := FALSE;
       "Q_Door_Open" := TRUE;
   END_IF;
   IF #_w1 AND "DB_Data".LS_Door_Opened THEN "Q_Door_Open" := FALSE; END_IF;
END_REGION

REGION Network 2: Nút nhấn MỞ cửa bên trong ca bin
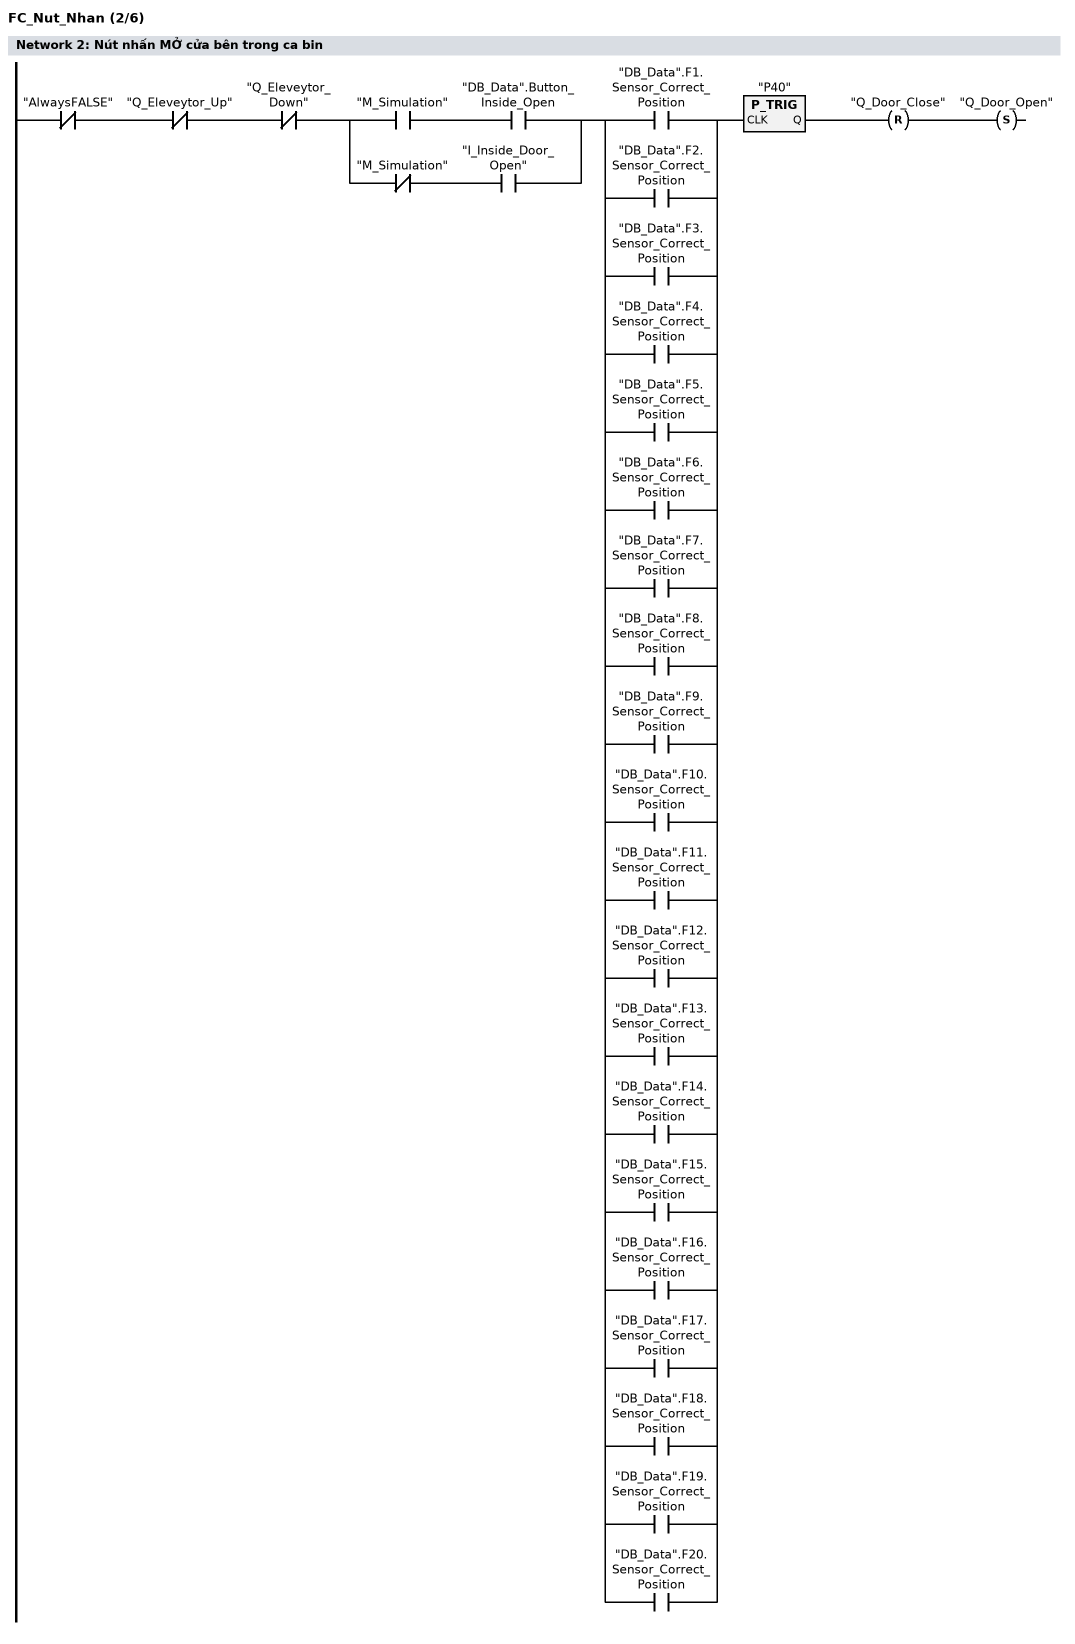
   RUNG wire#powerrail
      I_Contact( "AlwaysFALSE" )
      I_Contact( "Q_Eleveytor_Up" )
      I_Contact( "Q_Eleveytor_Down" )
      wire#w1
      Contact( "M_Simulation" )
      Contact( "DB_Data".Button_Inside_Open )
      wire#w2
      Contact( "DB_Data".F1.Sensor_Correct_Position )
      wire#w3
      P_Trig( "P40" )
      R_Coil( "Q_Door_Close" )
      S_Coil( "Q_Door_Open" )
   END_RUNG
   RUNG wire#w1
      I_Contact( "M_Simulation" )
      Contact( "I_Inside_Door_Open" )
   END_RUNG wire#w2
   RUNG wire#w2
      Contact( "DB_Data".F2.Sensor_Correct_Position )
   END_RUNG wire#w3
   RUNG wire#w2
      Contact( "DB_Data".F3.Sensor_Correct_Position )
   END_RUNG wire#w3
   RUNG wire#w2
      Contact( "DB_Data".F4.Sensor_Correct_Position )
   END_RUNG wire#w3
   RUNG wire#w2
      Contact( "DB_Data".F5.Sensor_Correct_Position )
   END_RUNG wire#w3
   RUNG wire#w2
      Contact( "DB_Data".F6.Sensor_Correct_Position )
   END_RUNG wire#w3
   RUNG wire#w2
      Contact( "DB_Data".F7.Sensor_Correct_Position )
   END_RUNG wire#w3
   RUNG wire#w2
      Contact( "DB_Data".F8.Sensor_Correct_Position )
   END_RUNG wire#w3
   RUNG wire#w2
      Contact( "DB_Data".F9.Sensor_Correct_Position )
   END_RUNG wire#w3
   RUNG wire#w2
      Contact( "DB_Data".F10.Sensor_Correct_Position )
   END_RUNG wire#w3
   RUNG wire#w2
      Contact( "DB_Data".F11.Sensor_Correct_Position )
   END_RUNG wire#w3
   RUNG wire#w2
      Contact( "DB_Data".F12.Sensor_Correct_Position )
   END_RUNG wire#w3
   RUNG wire#w2
      Contact( "DB_Data".F13.Sensor_Correct_Position )
   END_RUNG wire#w3
   RUNG wire#w2
      Contact( "DB_Data".F14.Sensor_Correct_Position )
   END_RUNG wire#w3
   RUNG wire#w2
      Contact( "DB_Data".F15.Sensor_Correct_Position )
   END_RUNG wire#w3
   RUNG wire#w2
      Contact( "DB_Data".F16.Sensor_Correct_Position )
   END_RUNG wire#w3
   RUNG wire#w2
      Contact( "DB_Data".F17.Sensor_Correct_Position )
   END_RUNG wire#w3
   RUNG wire#w2
      Contact( "DB_Data".F18.Sensor_Correct_Position )
   END_RUNG wire#w3
   RUNG wire#w2
      Contact( "DB_Data".F19.Sensor_Correct_Position )
   END_RUNG wire#w3
   RUNG wire#w2
      Contact( "DB_Data".F20.Sensor_Correct_Position )
   END_RUNG wire#w3
   // the same network as SCL:
   #_w1 := NOT "AlwaysFALSE" AND NOT "Q_Eleveytor_Up" AND NOT "Q_Eleveytor_Down" AND (("M_Simulation" AND "DB_Data".Button_Inside_Open) OR (NOT "M_Simulation" AND "I_Inside_Door_Open")) AND ("DB_Data".F1.Sensor_Correct_Position OR "DB_Data".F2.Sensor_Correct_Position OR "DB_Data".F3.Sensor_Correct_Position OR "DB_Data".F4.Sensor_Correct_Position OR "DB_Data".F5.Sensor_Correct_Position OR "DB_Data".F6.Sensor_Correct_Position OR "DB_Data".F7.Sensor_Correct_Position OR "DB_Data".F8.Sensor_Correct_Position OR "DB_Data".F9.Sensor_Correct_Position OR "DB_Data".F10.Sensor_Correct_Position OR "DB_Data".F11.Sensor_Correct_Position OR "DB_Data".F12.Sensor_Correct_Position OR "DB_Data".F13.Sensor_Correct_Position OR "DB_Data".F14.Sensor_Correct_Position OR "DB_Data".F15.Sensor_Correct_Position OR "DB_Data".F16.Sensor_Correct_Position OR "DB_Data".F17.Sensor_Correct_Position OR "DB_Data".F18.Sensor_Correct_Position OR "DB_Data".F19.Sensor_Correct_Position OR "DB_Data".F20.Sensor_Correct_Position);
   #_w2 := #_w1 AND NOT "P40";   // rising edge
   "P40" := #_w1;
   IF #_w2 THEN
       "Q_Door_Close" := FALSE;
       "Q_Door_Open" := TRUE;
   END_IF;
END_REGION

REGION Network 3: NÚT NHẤN ĐÓNG CỮA
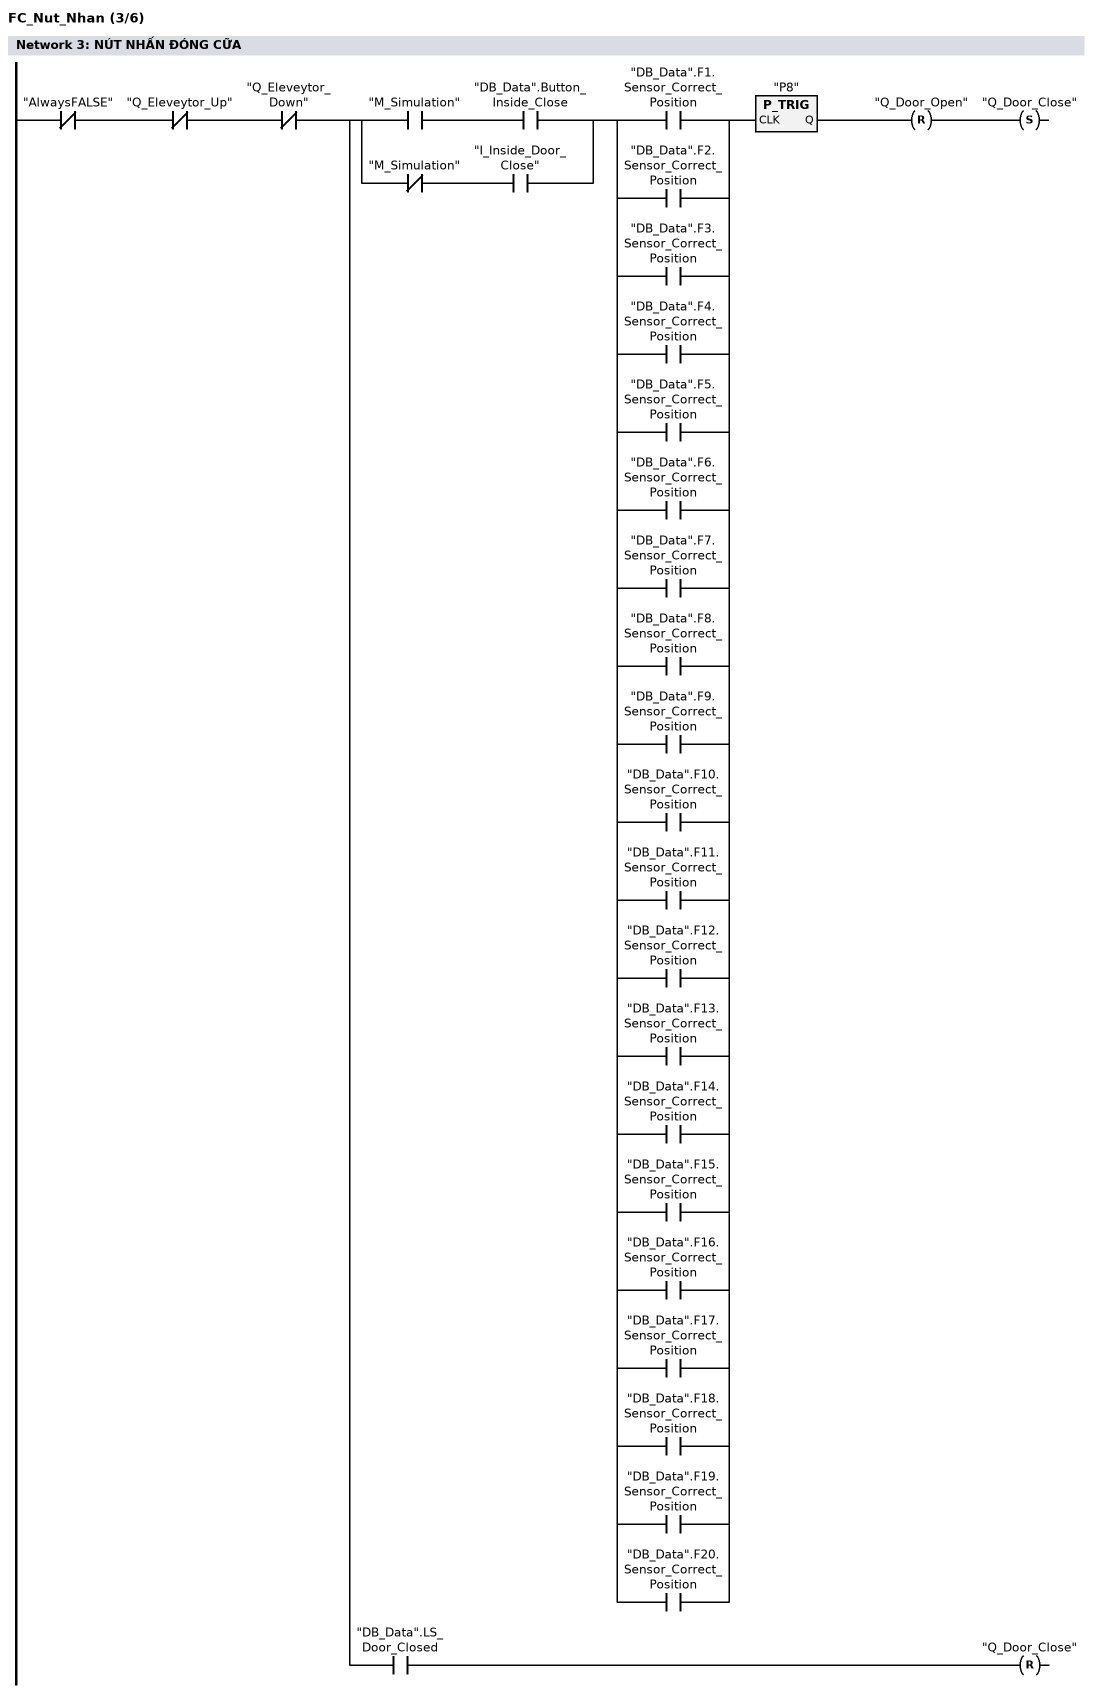
   RUNG wire#powerrail
      I_Contact( "AlwaysFALSE" )
      I_Contact( "Q_Eleveytor_Up" )
      I_Contact( "Q_Eleveytor_Down" )
      wire#w1
      Contact( "M_Simulation" )
      Contact( "DB_Data".Button_Inside_Close )
      wire#w2
      Contact( "DB_Data".F1.Sensor_Correct_Position )
      wire#w3
      P_Trig( "P8" )
      R_Coil( "Q_Door_Open" )
      S_Coil( "Q_Door_Close" )
   END_RUNG
   RUNG wire#w1
      I_Contact( "M_Simulation" )
      Contact( "I_Inside_Door_Close" )
   END_RUNG wire#w2
   RUNG wire#w2
      Contact( "DB_Data".F2.Sensor_Correct_Position )
   END_RUNG wire#w3
   RUNG wire#w2
      Contact( "DB_Data".F3.Sensor_Correct_Position )
   END_RUNG wire#w3
   RUNG wire#w2
      Contact( "DB_Data".F4.Sensor_Correct_Position )
   END_RUNG wire#w3
   RUNG wire#w2
      Contact( "DB_Data".F5.Sensor_Correct_Position )
   END_RUNG wire#w3
   RUNG wire#w2
      Contact( "DB_Data".F6.Sensor_Correct_Position )
   END_RUNG wire#w3
   RUNG wire#w2
      Contact( "DB_Data".F7.Sensor_Correct_Position )
   END_RUNG wire#w3
   RUNG wire#w2
      Contact( "DB_Data".F8.Sensor_Correct_Position )
   END_RUNG wire#w3
   RUNG wire#w2
      Contact( "DB_Data".F9.Sensor_Correct_Position )
   END_RUNG wire#w3
   RUNG wire#w2
      Contact( "DB_Data".F10.Sensor_Correct_Position )
   END_RUNG wire#w3
   RUNG wire#w2
      Contact( "DB_Data".F11.Sensor_Correct_Position )
   END_RUNG wire#w3
   RUNG wire#w2
      Contact( "DB_Data".F12.Sensor_Correct_Position )
   END_RUNG wire#w3
   RUNG wire#w2
      Contact( "DB_Data".F13.Sensor_Correct_Position )
   END_RUNG wire#w3
   RUNG wire#w2
      Contact( "DB_Data".F14.Sensor_Correct_Position )
   END_RUNG wire#w3
   RUNG wire#w2
      Contact( "DB_Data".F15.Sensor_Correct_Position )
   END_RUNG wire#w3
   RUNG wire#w2
      Contact( "DB_Data".F16.Sensor_Correct_Position )
   END_RUNG wire#w3
   RUNG wire#w2
      Contact( "DB_Data".F17.Sensor_Correct_Position )
   END_RUNG wire#w3
   RUNG wire#w2
      Contact( "DB_Data".F18.Sensor_Correct_Position )
   END_RUNG wire#w3
   RUNG wire#w2
      Contact( "DB_Data".F19.Sensor_Correct_Position )
   END_RUNG wire#w3
   RUNG wire#w2
      Contact( "DB_Data".F20.Sensor_Correct_Position )
   END_RUNG wire#w3
   RUNG wire#w1
      Contact( "DB_Data".LS_Door_Closed )
      R_Coil( "Q_Door_Close" )
   END_RUNG
   // the same network as SCL:
   #_w1 := NOT "AlwaysFALSE" AND NOT "Q_Eleveytor_Up" AND NOT "Q_Eleveytor_Down";
   #_w2 := #_w1 AND (("M_Simulation" AND "DB_Data".Button_Inside_Close) OR (NOT "M_Simulation" AND "I_Inside_Door_Close")) AND ("DB_Data".F1.Sensor_Correct_Position OR "DB_Data".F2.Sensor_Correct_Position OR "DB_Data".F3.Sensor_Correct_Position OR "DB_Data".F4.Sensor_Correct_Position OR "DB_Data".F5.Sensor_Correct_Position OR "DB_Data".F6.Sensor_Correct_Position OR "DB_Data".F7.Sensor_Correct_Position OR "DB_Data".F8.Sensor_Correct_Position OR "DB_Data".F9.Sensor_Correct_Position OR "DB_Data".F10.Sensor_Correct_Position OR "DB_Data".F11.Sensor_Correct_Position OR "DB_Data".F12.Sensor_Correct_Position OR "DB_Data".F13.Sensor_Correct_Position OR "DB_Data".F14.Sensor_Correct_Position OR "DB_Data".F15.Sensor_Correct_Position OR "DB_Data".F16.Sensor_Correct_Position OR "DB_Data".F17.Sensor_Correct_Position OR "DB_Data".F18.Sensor_Correct_Position OR "DB_Data".F19.Sensor_Correct_Position OR "DB_Data".F20.Sensor_Correct_Position);
   #_w3 := #_w2 AND NOT "P8";   // rising edge
   "P8" := #_w2;
   IF #_w3 THEN
       "Q_Door_Open" := FALSE;
       "Q_Door_Close" := TRUE;
   END_IF;
   IF #_w1 AND "DB_Data".LS_Door_Closed THEN "Q_Door_Close" := FALSE; END_IF;
END_REGION

REGION Network 4: Nút nhấn chọn tầng tại các tầng
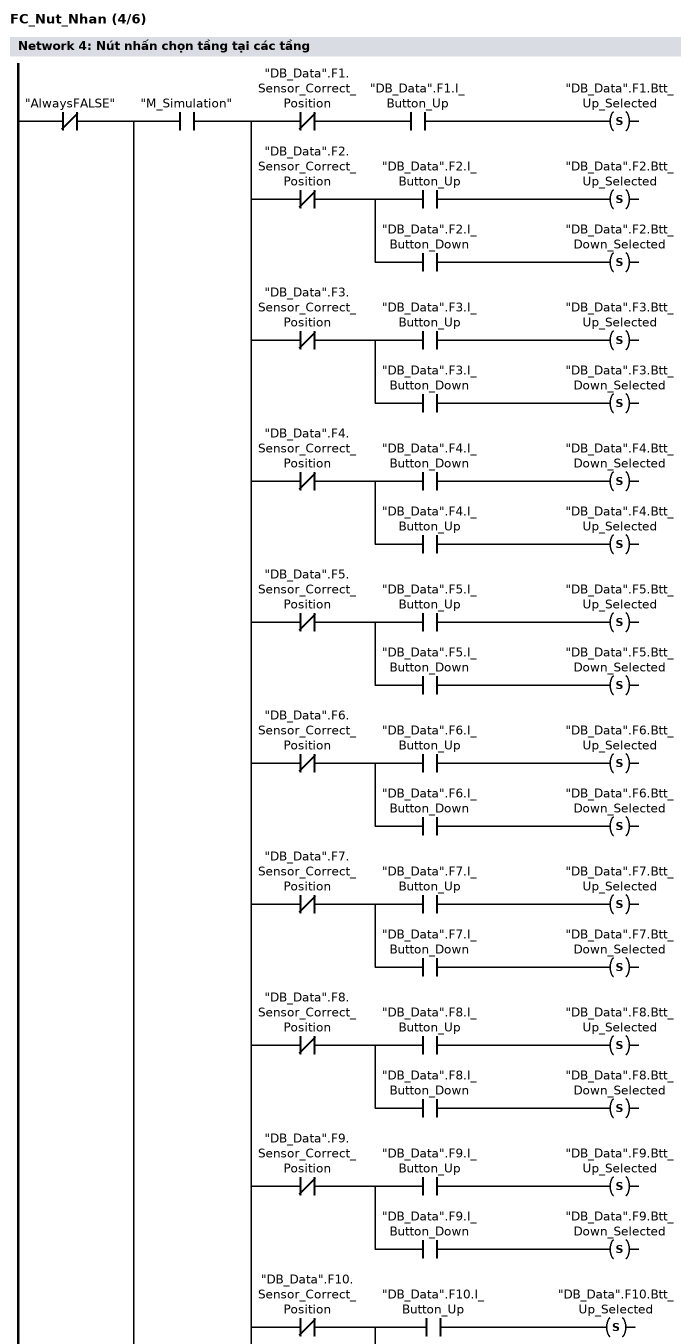
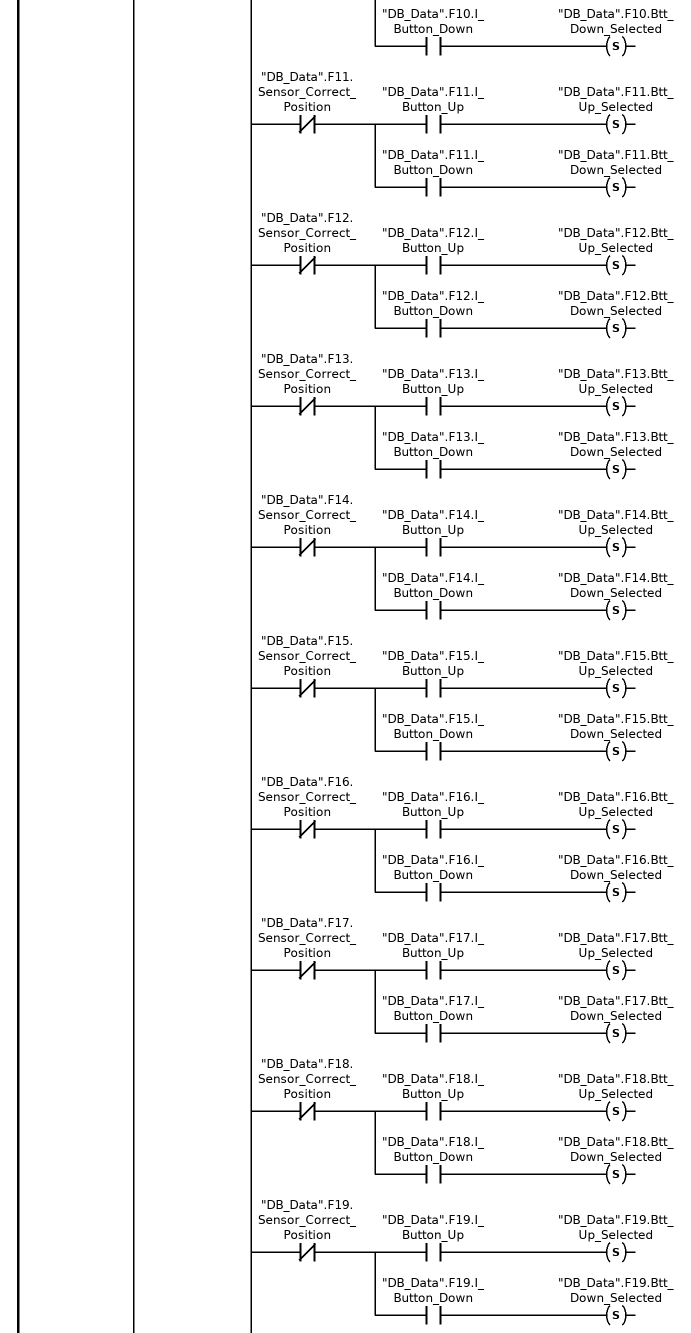
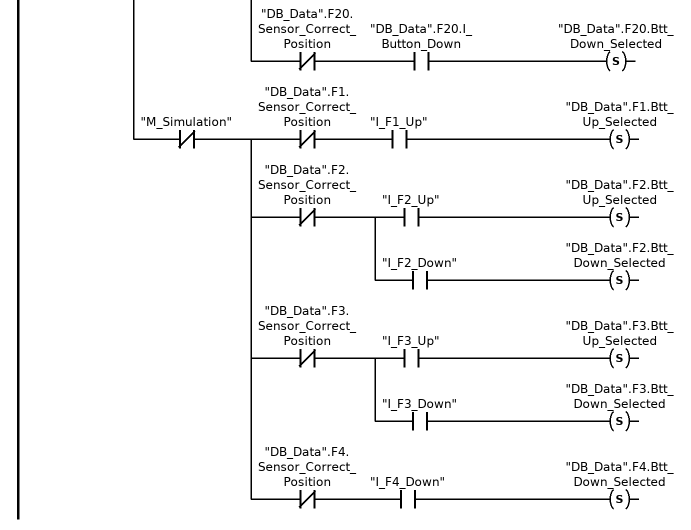
   RUNG wire#powerrail
      I_Contact( "AlwaysFALSE" )
      wire#w1
      Contact( "M_Simulation" )
      wire#w2
      I_Contact( "DB_Data".F1.Sensor_Correct_Position )
      Contact( "DB_Data".F1.I_Button_Up )
      S_Coil( "DB_Data".F1.Btt_Up_Selected )
   END_RUNG
   RUNG wire#w2
      I_Contact( "DB_Data".F2.Sensor_Correct_Position )
      wire#w3
      Contact( "DB_Data".F2.I_Button_Up )
      S_Coil( "DB_Data".F2.Btt_Up_Selected )
   END_RUNG
   RUNG wire#w3
      Contact( "DB_Data".F2.I_Button_Down )
      S_Coil( "DB_Data".F2.Btt_Down_Selected )
   END_RUNG
   RUNG wire#w2
      I_Contact( "DB_Data".F3.Sensor_Correct_Position )
      wire#w4
      Contact( "DB_Data".F3.I_Button_Up )
      S_Coil( "DB_Data".F3.Btt_Up_Selected )
   END_RUNG
   RUNG wire#w4
      Contact( "DB_Data".F3.I_Button_Down )
      S_Coil( "DB_Data".F3.Btt_Down_Selected )
   END_RUNG
   RUNG wire#w2
      I_Contact( "DB_Data".F4.Sensor_Correct_Position )
      wire#w5
      Contact( "DB_Data".F4.I_Button_Down )
      S_Coil( "DB_Data".F4.Btt_Down_Selected )
   END_RUNG
   RUNG wire#w5
      Contact( "DB_Data".F4.I_Button_Up )
      S_Coil( "DB_Data".F4.Btt_Up_Selected )
   END_RUNG
   RUNG wire#w2
      I_Contact( "DB_Data".F5.Sensor_Correct_Position )
      wire#w6
      Contact( "DB_Data".F5.I_Button_Up )
      S_Coil( "DB_Data".F5.Btt_Up_Selected )
   END_RUNG
   RUNG wire#w6
      Contact( "DB_Data".F5.I_Button_Down )
      S_Coil( "DB_Data".F5.Btt_Down_Selected )
   END_RUNG
   RUNG wire#w2
      I_Contact( "DB_Data".F6.Sensor_Correct_Position )
      wire#w7
      Contact( "DB_Data".F6.I_Button_Up )
      S_Coil( "DB_Data".F6.Btt_Up_Selected )
   END_RUNG
   RUNG wire#w7
      Contact( "DB_Data".F6.I_Button_Down )
      S_Coil( "DB_Data".F6.Btt_Down_Selected )
   END_RUNG
   RUNG wire#w2
      I_Contact( "DB_Data".F7.Sensor_Correct_Position )
      wire#w8
      Contact( "DB_Data".F7.I_Button_Up )
      S_Coil( "DB_Data".F7.Btt_Up_Selected )
   END_RUNG
   RUNG wire#w8
      Contact( "DB_Data".F7.I_Button_Down )
      S_Coil( "DB_Data".F7.Btt_Down_Selected )
   END_RUNG
   RUNG wire#w2
      I_Contact( "DB_Data".F8.Sensor_Correct_Position )
      wire#w9
      Contact( "DB_Data".F8.I_Button_Up )
      S_Coil( "DB_Data".F8.Btt_Up_Selected )
   END_RUNG
   RUNG wire#w9
      Contact( "DB_Data".F8.I_Button_Down )
      S_Coil( "DB_Data".F8.Btt_Down_Selected )
   END_RUNG
   RUNG wire#w2
      I_Contact( "DB_Data".F9.Sensor_Correct_Position )
      wire#w10
      Contact( "DB_Data".F9.I_Button_Up )
      S_Coil( "DB_Data".F9.Btt_Up_Selected )
   END_RUNG
   RUNG wire#w10
      Contact( "DB_Data".F9.I_Button_Down )
      S_Coil( "DB_Data".F9.Btt_Down_Selected )
   END_RUNG
   RUNG wire#w2
      I_Contact( "DB_Data".F10.Sensor_Correct_Position )
      wire#w11
      Contact( "DB_Data".F10.I_Button_Up )
      S_Coil( "DB_Data".F10.Btt_Up_Selected )
   END_RUNG
   RUNG wire#w11
      Contact( "DB_Data".F10.I_Button_Down )
      S_Coil( "DB_Data".F10.Btt_Down_Selected )
   END_RUNG
   RUNG wire#w2
      I_Contact( "DB_Data".F11.Sensor_Correct_Position )
      wire#w12
      Contact( "DB_Data".F11.I_Button_Up )
      S_Coil( "DB_Data".F11.Btt_Up_Selected )
   END_RUNG
   RUNG wire#w12
      Contact( "DB_Data".F11.I_Button_Down )
      S_Coil( "DB_Data".F11.Btt_Down_Selected )
   END_RUNG
   RUNG wire#w2
      I_Contact( "DB_Data".F12.Sensor_Correct_Position )
      wire#w13
      Contact( "DB_Data".F12.I_Button_Up )
      S_Coil( "DB_Data".F12.Btt_Up_Selected )
   END_RUNG
   RUNG wire#w13
      Contact( "DB_Data".F12.I_Button_Down )
      S_Coil( "DB_Data".F12.Btt_Down_Selected )
   END_RUNG
   RUNG wire#w2
      I_Contact( "DB_Data".F13.Sensor_Correct_Position )
      wire#w14
      Contact( "DB_Data".F13.I_Button_Up )
      S_Coil( "DB_Data".F13.Btt_Up_Selected )
   END_RUNG
   RUNG wire#w14
      Contact( "DB_Data".F13.I_Button_Down )
      S_Coil( "DB_Data".F13.Btt_Down_Selected )
   END_RUNG
   RUNG wire#w2
      I_Contact( "DB_Data".F14.Sensor_Correct_Position )
      wire#w15
      Contact( "DB_Data".F14.I_Button_Up )
      S_Coil( "DB_Data".F14.Btt_Up_Selected )
   END_RUNG
   RUNG wire#w15
      Contact( "DB_Data".F14.I_Button_Down )
      S_Coil( "DB_Data".F14.Btt_Down_Selected )
   END_RUNG
   RUNG wire#w2
      I_Contact( "DB_Data".F15.Sensor_Correct_Position )
      wire#w16
      Contact( "DB_Data".F15.I_Button_Up )
      S_Coil( "DB_Data".F15.Btt_Up_Selected )
   END_RUNG
   RUNG wire#w16
      Contact( "DB_Data".F15.I_Button_Down )
      S_Coil( "DB_Data".F15.Btt_Down_Selected )
   END_RUNG
   RUNG wire#w2
      I_Contact( "DB_Data".F16.Sensor_Correct_Position )
      wire#w17
      Contact( "DB_Data".F16.I_Button_Up )
      S_Coil( "DB_Data".F16.Btt_Up_Selected )
   END_RUNG
   RUNG wire#w17
      Contact( "DB_Data".F16.I_Button_Down )
      S_Coil( "DB_Data".F16.Btt_Down_Selected )
   END_RUNG
   RUNG wire#w2
      I_Contact( "DB_Data".F17.Sensor_Correct_Position )
      wire#w18
      Contact( "DB_Data".F17.I_Button_Up )
      S_Coil( "DB_Data".F17.Btt_Up_Selected )
   END_RUNG
   RUNG wire#w18
      Contact( "DB_Data".F17.I_Button_Down )
      S_Coil( "DB_Data".F17.Btt_Down_Selected )
   END_RUNG
   RUNG wire#w2
      I_Contact( "DB_Data".F18.Sensor_Correct_Position )
      wire#w19
      Contact( "DB_Data".F18.I_Button_Up )
      S_Coil( "DB_Data".F18.Btt_Up_Selected )
   END_RUNG
   RUNG wire#w19
      Contact( "DB_Data".F18.I_Button_Down )
      S_Coil( "DB_Data".F18.Btt_Down_Selected )
   END_RUNG
   RUNG wire#w2
      I_Contact( "DB_Data".F19.Sensor_Correct_Position )
      wire#w20
      Contact( "DB_Data".F19.I_Button_Up )
      S_Coil( "DB_Data".F19.Btt_Up_Selected )
   END_RUNG
   RUNG wire#w20
      Contact( "DB_Data".F19.I_Button_Down )
      S_Coil( "DB_Data".F19.Btt_Down_Selected )
   END_RUNG
   RUNG wire#w2
      I_Contact( "DB_Data".F20.Sensor_Correct_Position )
      Contact( "DB_Data".F20.I_Button_Down )
      S_Coil( "DB_Data".F20.Btt_Down_Selected )
   END_RUNG
   RUNG wire#w1
      I_Contact( "M_Simulation" )
      wire#w21
      I_Contact( "DB_Data".F1.Sensor_Correct_Position )
      Contact( "I_F1_Up" )
      S_Coil( "DB_Data".F1.Btt_Up_Selected )
   END_RUNG
   RUNG wire#w21
      I_Contact( "DB_Data".F2.Sensor_Correct_Position )
      wire#w22
      Contact( "I_F2_Up" )
      S_Coil( "DB_Data".F2.Btt_Up_Selected )
   END_RUNG
   RUNG wire#w22
      Contact( "I_F2_Down" )
      S_Coil( "DB_Data".F2.Btt_Down_Selected )
   END_RUNG
   RUNG wire#w21
      I_Contact( "DB_Data".F3.Sensor_Correct_Position )
      wire#w23
      Contact( "I_F3_Up" )
      S_Coil( "DB_Data".F3.Btt_Up_Selected )
   END_RUNG
   RUNG wire#w23
      Contact( "I_F3_Down" )
      S_Coil( "DB_Data".F3.Btt_Down_Selected )
   END_RUNG
   RUNG wire#w21
      I_Contact( "DB_Data".F4.Sensor_Correct_Position )
      Contact( "I_F4_Down" )
      S_Coil( "DB_Data".F4.Btt_Down_Selected )
   END_RUNG
   // the same network as SCL:
   #_w1 := NOT "AlwaysFALSE" AND "M_Simulation";
   IF #_w1 AND NOT "DB_Data".F1.Sensor_Correct_Position AND "DB_Data".F1.I_Button_Up THEN
       "DB_Data".F1.Btt_Up_Selected := TRUE;
   END_IF;
   #_w2 := #_w1 AND NOT "DB_Data".F2.Sensor_Correct_Position;
   IF #_w2 AND "DB_Data".F2.I_Button_Up THEN "DB_Data".F2.Btt_Up_Selected := TRUE; END_IF;
   IF #_w2 AND "DB_Data".F2.I_Button_Down THEN "DB_Data".F2.Btt_Down_Selected := TRUE; END_IF;
   #_w3 := #_w1 AND NOT "DB_Data".F3.Sensor_Correct_Position;
   IF #_w3 AND "DB_Data".F3.I_Button_Up THEN "DB_Data".F3.Btt_Up_Selected := TRUE; END_IF;
   IF #_w3 AND "DB_Data".F3.I_Button_Down THEN "DB_Data".F3.Btt_Down_Selected := TRUE; END_IF;
   #_w4 := #_w1 AND NOT "DB_Data".F4.Sensor_Correct_Position;
   IF #_w4 AND "DB_Data".F4.I_Button_Down THEN "DB_Data".F4.Btt_Down_Selected := TRUE; END_IF;
   IF #_w4 AND "DB_Data".F4.I_Button_Up THEN "DB_Data".F4.Btt_Up_Selected := TRUE; END_IF;
   #_w5 := #_w1 AND NOT "DB_Data".F5.Sensor_Correct_Position;
   IF #_w5 AND "DB_Data".F5.I_Button_Up THEN "DB_Data".F5.Btt_Up_Selected := TRUE; END_IF;
   IF #_w5 AND "DB_Data".F5.I_Button_Down THEN "DB_Data".F5.Btt_Down_Selected := TRUE; END_IF;
   #_w6 := #_w1 AND NOT "DB_Data".F6.Sensor_Correct_Position;
   IF #_w6 AND "DB_Data".F6.I_Button_Up THEN "DB_Data".F6.Btt_Up_Selected := TRUE; END_IF;
   IF #_w6 AND "DB_Data".F6.I_Button_Down THEN "DB_Data".F6.Btt_Down_Selected := TRUE; END_IF;
   #_w7 := #_w1 AND NOT "DB_Data".F7.Sensor_Correct_Position;
   IF #_w7 AND "DB_Data".F7.I_Button_Up THEN "DB_Data".F7.Btt_Up_Selected := TRUE; END_IF;
   IF #_w7 AND "DB_Data".F7.I_Button_Down THEN "DB_Data".F7.Btt_Down_Selected := TRUE; END_IF;
   #_w8 := #_w1 AND NOT "DB_Data".F8.Sensor_Correct_Position;
   IF #_w8 AND "DB_Data".F8.I_Button_Up THEN "DB_Data".F8.Btt_Up_Selected := TRUE; END_IF;
   IF #_w8 AND "DB_Data".F8.I_Button_Down THEN "DB_Data".F8.Btt_Down_Selected := TRUE; END_IF;
   #_w9 := #_w1 AND NOT "DB_Data".F9.Sensor_Correct_Position;
   IF #_w9 AND "DB_Data".F9.I_Button_Up THEN "DB_Data".F9.Btt_Up_Selected := TRUE; END_IF;
   IF #_w9 AND "DB_Data".F9.I_Button_Down THEN "DB_Data".F9.Btt_Down_Selected := TRUE; END_IF;
   #_w10 := #_w1 AND NOT "DB_Data".F10.Sensor_Correct_Position;
   IF #_w10 AND "DB_Data".F10.I_Button_Up THEN "DB_Data".F10.Btt_Up_Selected := TRUE; END_IF;
   IF #_w10 AND "DB_Data".F10.I_Button_Down THEN "DB_Data".F10.Btt_Down_Selected := TRUE; END_IF;
   #_w11 := #_w1 AND NOT "DB_Data".F11.Sensor_Correct_Position;
   IF #_w11 AND "DB_Data".F11.I_Button_Up THEN "DB_Data".F11.Btt_Up_Selected := TRUE; END_IF;
   IF #_w11 AND "DB_Data".F11.I_Button_Down THEN "DB_Data".F11.Btt_Down_Selected := TRUE; END_IF;
   #_w12 := #_w1 AND NOT "DB_Data".F12.Sensor_Correct_Position;
   IF #_w12 AND "DB_Data".F12.I_Button_Up THEN "DB_Data".F12.Btt_Up_Selected := TRUE; END_IF;
   IF #_w12 AND "DB_Data".F12.I_Button_Down THEN "DB_Data".F12.Btt_Down_Selected := TRUE; END_IF;
   #_w13 := #_w1 AND NOT "DB_Data".F13.Sensor_Correct_Position;
   IF #_w13 AND "DB_Data".F13.I_Button_Up THEN "DB_Data".F13.Btt_Up_Selected := TRUE; END_IF;
   IF #_w13 AND "DB_Data".F13.I_Button_Down THEN "DB_Data".F13.Btt_Down_Selected := TRUE; END_IF;
   #_w14 := #_w1 AND NOT "DB_Data".F14.Sensor_Correct_Position;
   IF #_w14 AND "DB_Data".F14.I_Button_Up THEN "DB_Data".F14.Btt_Up_Selected := TRUE; END_IF;
   IF #_w14 AND "DB_Data".F14.I_Button_Down THEN "DB_Data".F14.Btt_Down_Selected := TRUE; END_IF;
   #_w15 := #_w1 AND NOT "DB_Data".F15.Sensor_Correct_Position;
   IF #_w15 AND "DB_Data".F15.I_Button_Up THEN "DB_Data".F15.Btt_Up_Selected := TRUE; END_IF;
   IF #_w15 AND "DB_Data".F15.I_Button_Down THEN "DB_Data".F15.Btt_Down_Selected := TRUE; END_IF;
   #_w16 := #_w1 AND NOT "DB_Data".F16.Sensor_Correct_Position;
   IF #_w16 AND "DB_Data".F16.I_Button_Up THEN "DB_Data".F16.Btt_Up_Selected := TRUE; END_IF;
   IF #_w16 AND "DB_Data".F16.I_Button_Down THEN "DB_Data".F16.Btt_Down_Selected := TRUE; END_IF;
   #_w17 := #_w1 AND NOT "DB_Data".F17.Sensor_Correct_Position;
   IF #_w17 AND "DB_Data".F17.I_Button_Up THEN "DB_Data".F17.Btt_Up_Selected := TRUE; END_IF;
   IF #_w17 AND "DB_Data".F17.I_Button_Down THEN "DB_Data".F17.Btt_Down_Selected := TRUE; END_IF;
   #_w18 := #_w1 AND NOT "DB_Data".F18.Sensor_Correct_Position;
   IF #_w18 AND "DB_Data".F18.I_Button_Up THEN "DB_Data".F18.Btt_Up_Selected := TRUE; END_IF;
   IF #_w18 AND "DB_Data".F18.I_Button_Down THEN "DB_Data".F18.Btt_Down_Selected := TRUE; END_IF;
   #_w19 := #_w1 AND NOT "DB_Data".F19.Sensor_Correct_Position;
   IF #_w19 AND "DB_Data".F19.I_Button_Up THEN "DB_Data".F19.Btt_Up_Selected := TRUE; END_IF;
   IF #_w19 AND "DB_Data".F19.I_Button_Down THEN "DB_Data".F19.Btt_Down_Selected := TRUE; END_IF;
   IF #_w1 AND NOT "DB_Data".F20.Sensor_Correct_Position AND "DB_Data".F20.I_Button_Down THEN
       "DB_Data".F20.Btt_Down_Selected := TRUE;
   END_IF;
   #_w20 := NOT "AlwaysFALSE" AND NOT "M_Simulation";
   IF #_w20 AND NOT "DB_Data".F1.Sensor_Correct_Position AND "I_F1_Up" THEN
       "DB_Data".F1.Btt_Up_Selected := TRUE;
   END_IF;
   #_w21 := #_w20 AND NOT "DB_Data".F2.Sensor_Correct_Position;
   IF #_w21 AND "I_F2_Up" THEN "DB_Data".F2.Btt_Up_Selected := TRUE; END_IF;
   IF #_w21 AND "I_F2_Down" THEN "DB_Data".F2.Btt_Down_Selected := TRUE; END_IF;
   #_w22 := #_w20 AND NOT "DB_Data".F3.Sensor_Correct_Position;
   IF #_w22 AND "I_F3_Up" THEN "DB_Data".F3.Btt_Up_Selected := TRUE; END_IF;
   IF #_w22 AND "I_F3_Down" THEN "DB_Data".F3.Btt_Down_Selected := TRUE; END_IF;
   IF #_w20 AND NOT "DB_Data".F4.Sensor_Correct_Position AND "I_F4_Down" THEN
       "DB_Data".F4.Btt_Down_Selected := TRUE;
   END_IF;
END_REGION

REGION Network 5: Nút nhấn chọn tầng trong buồng thang
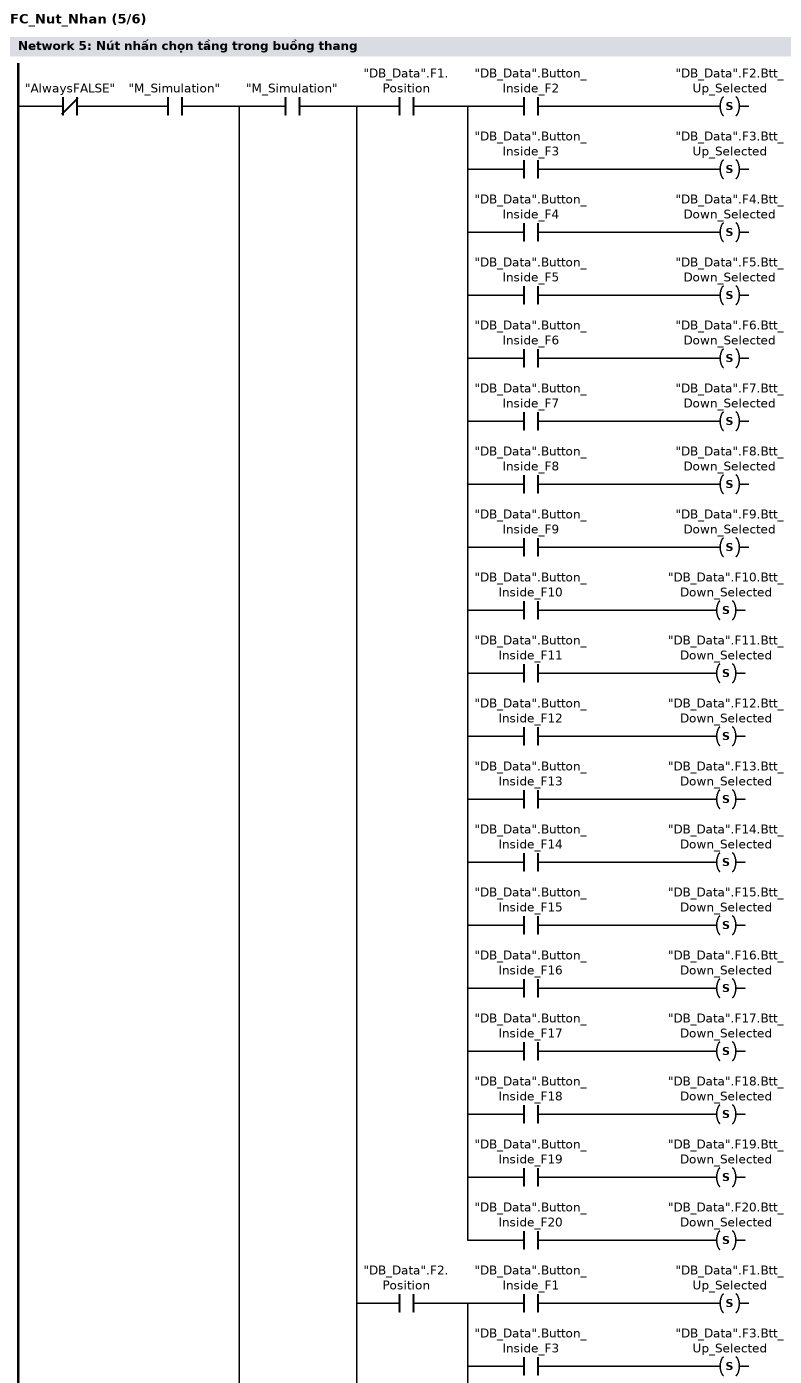
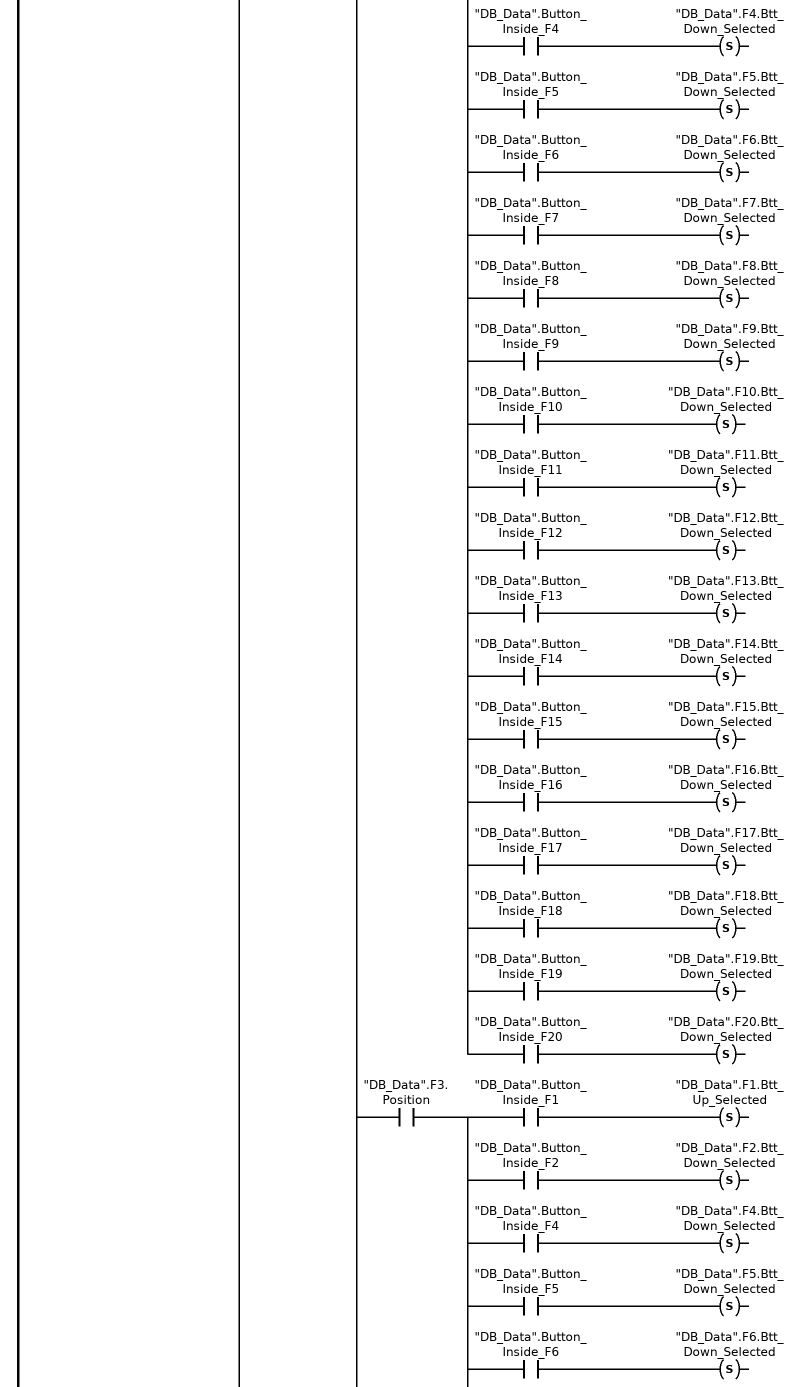
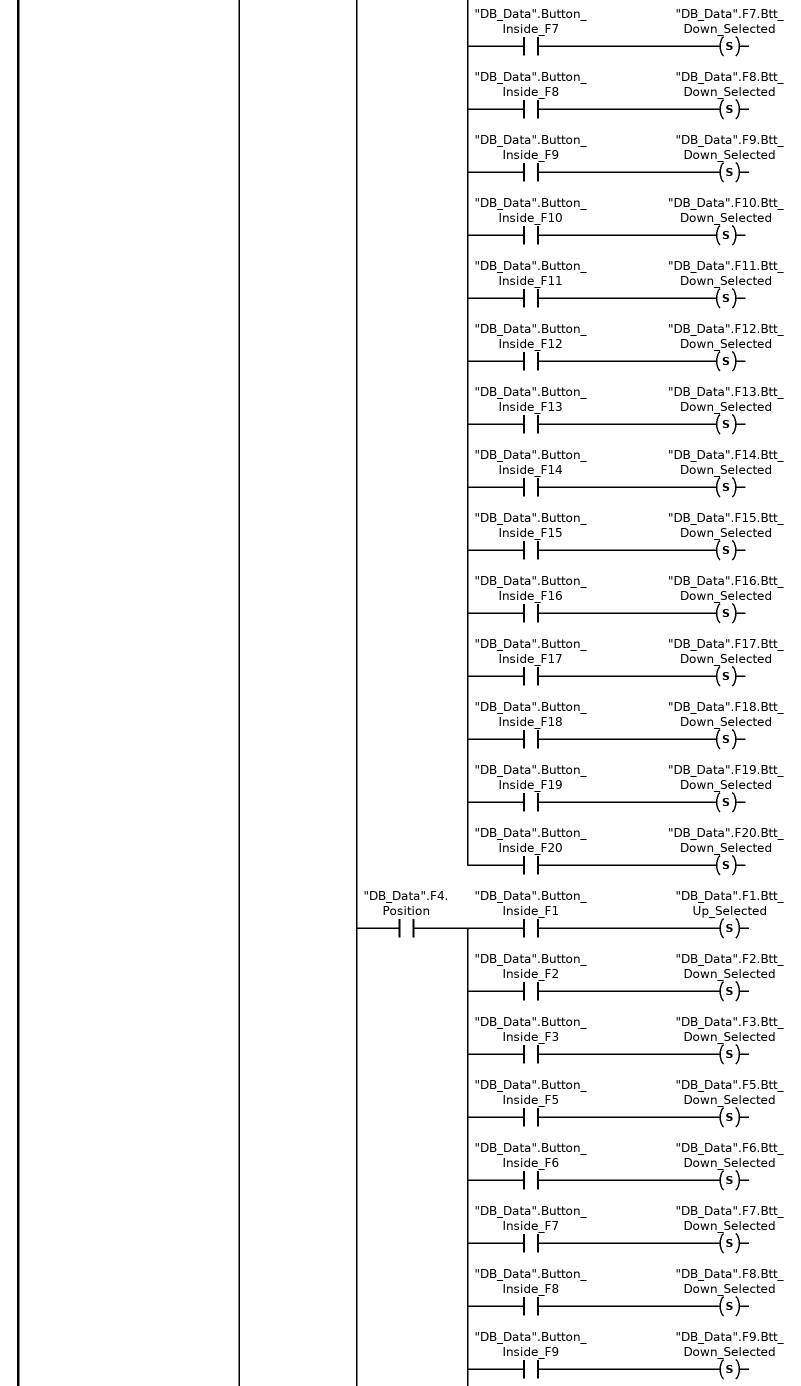
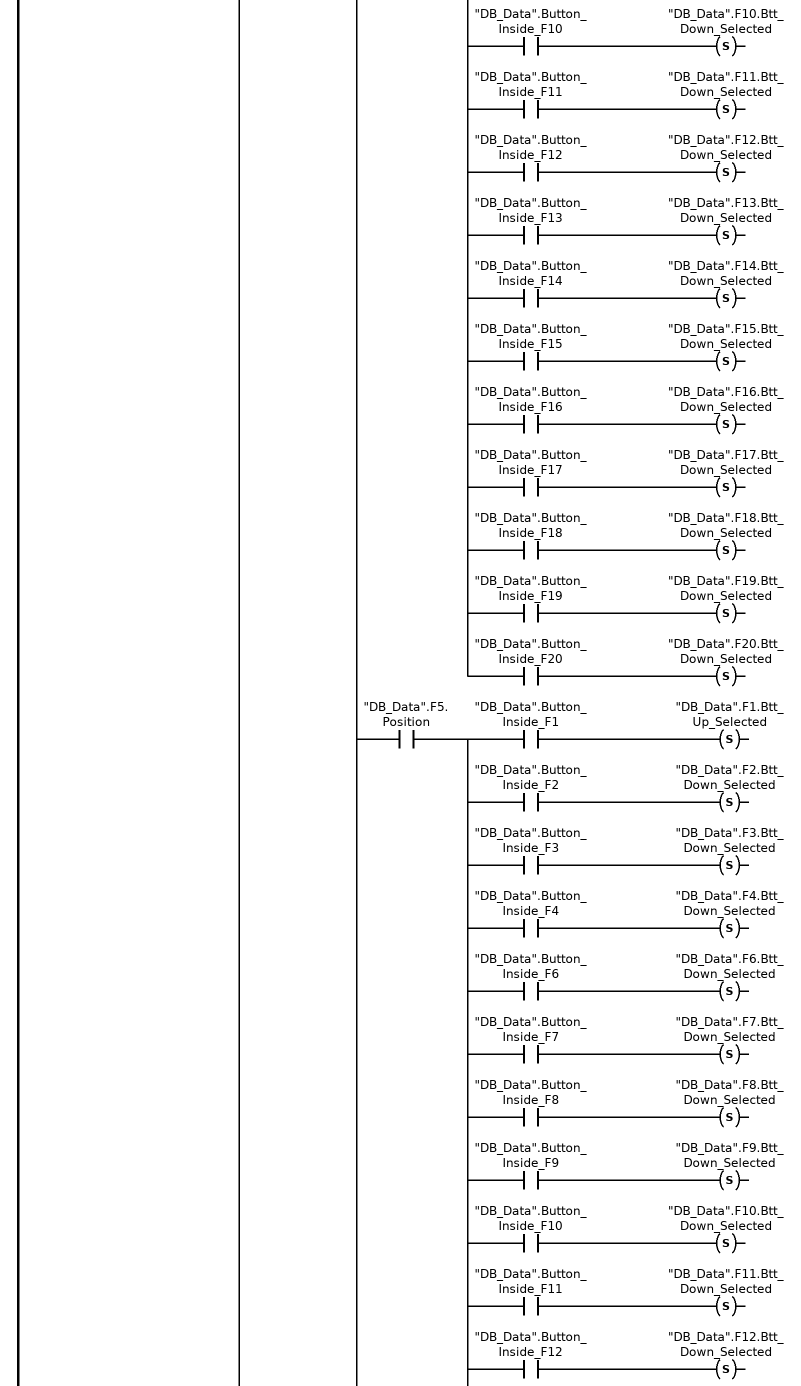
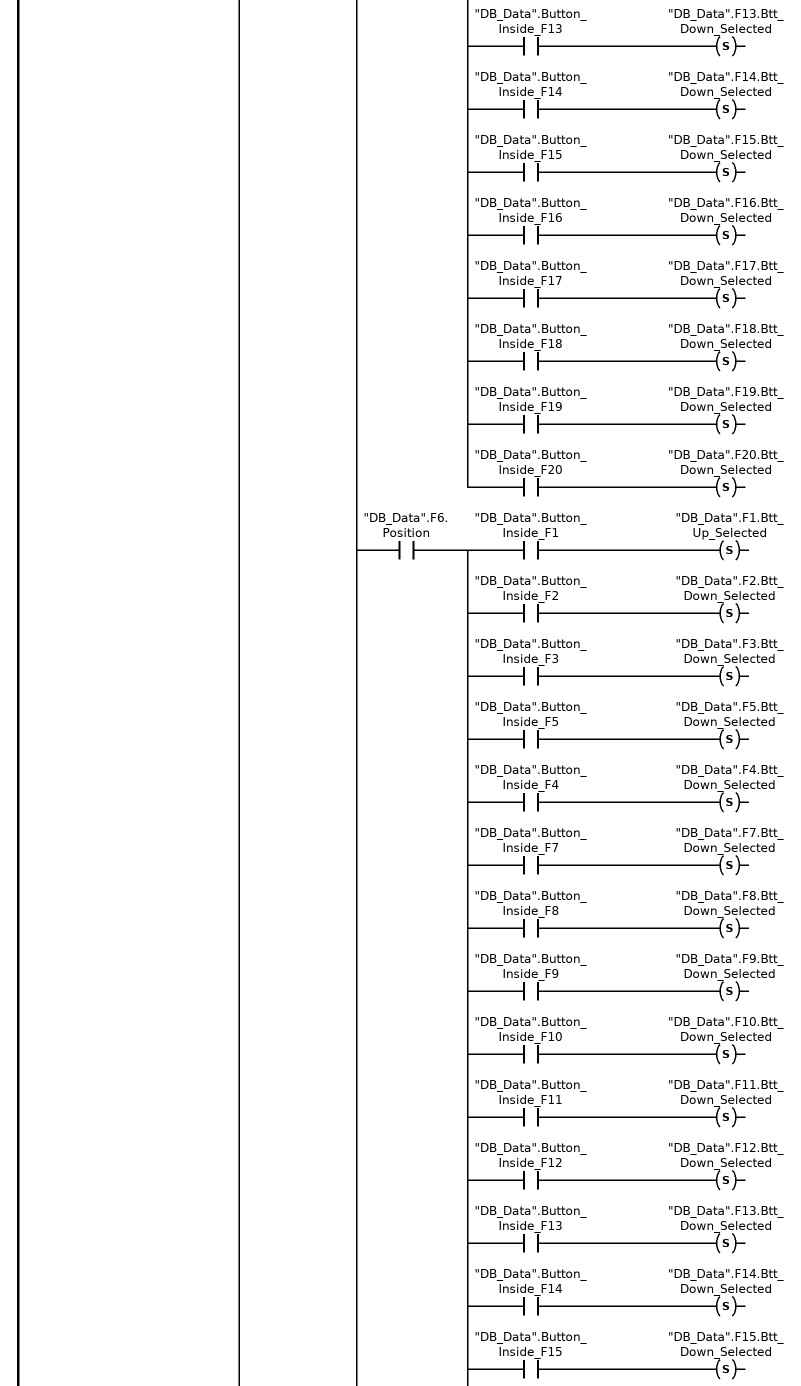
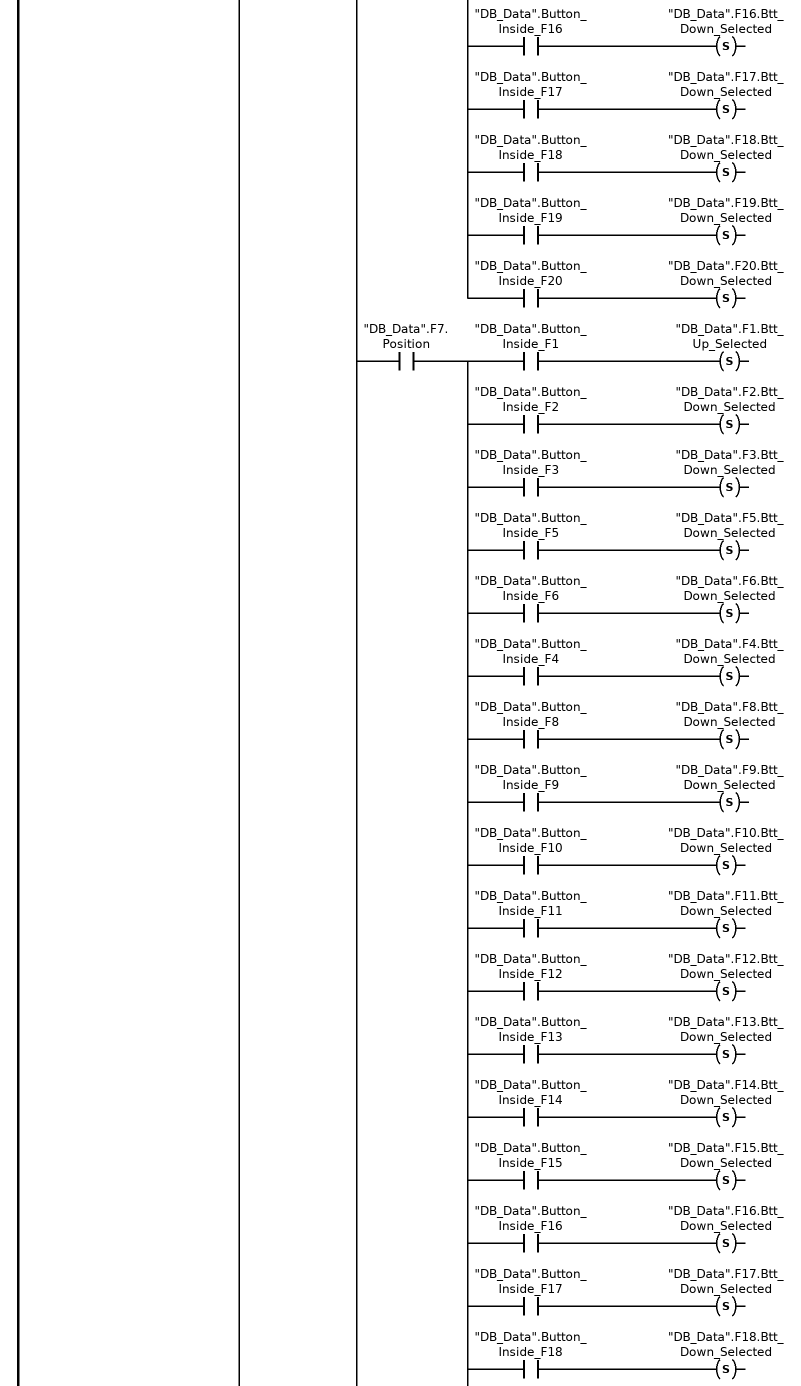
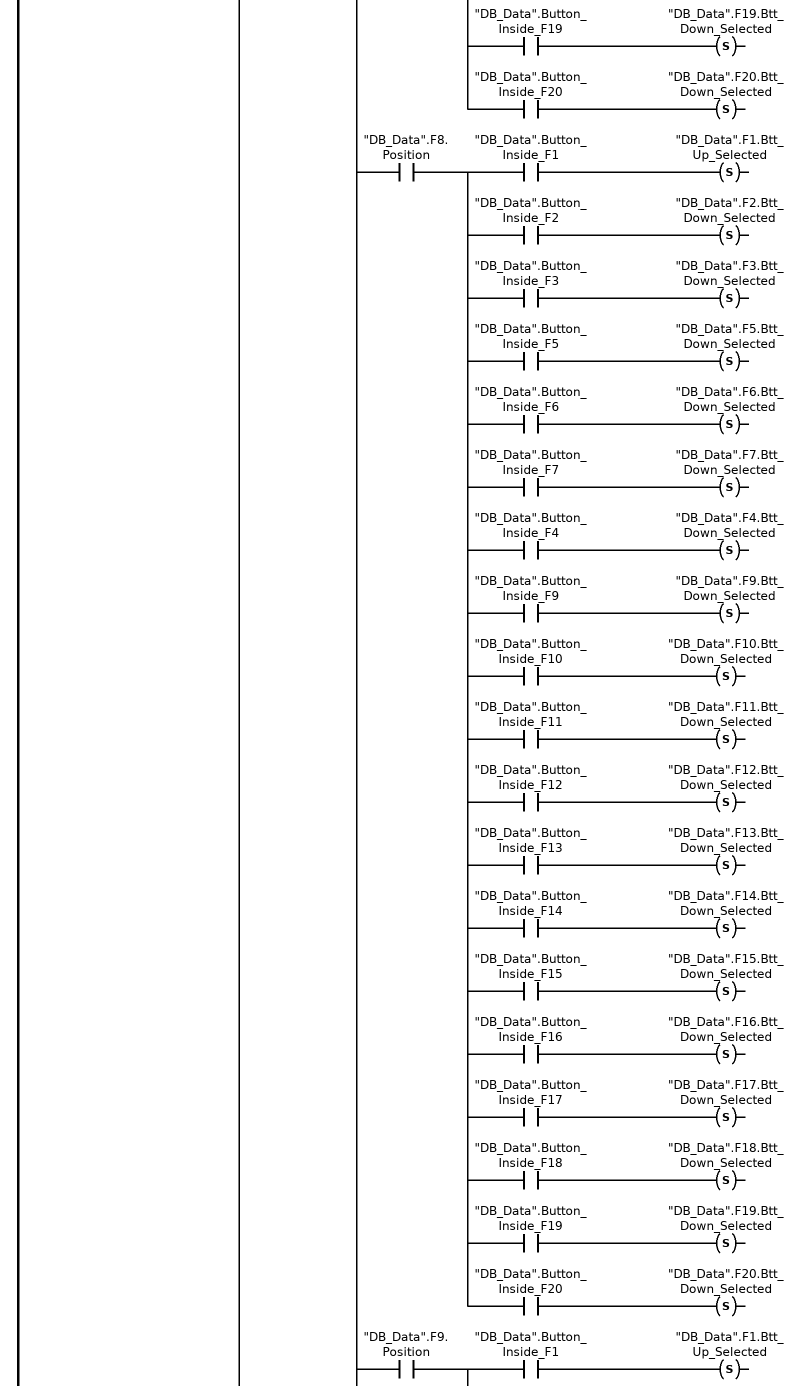
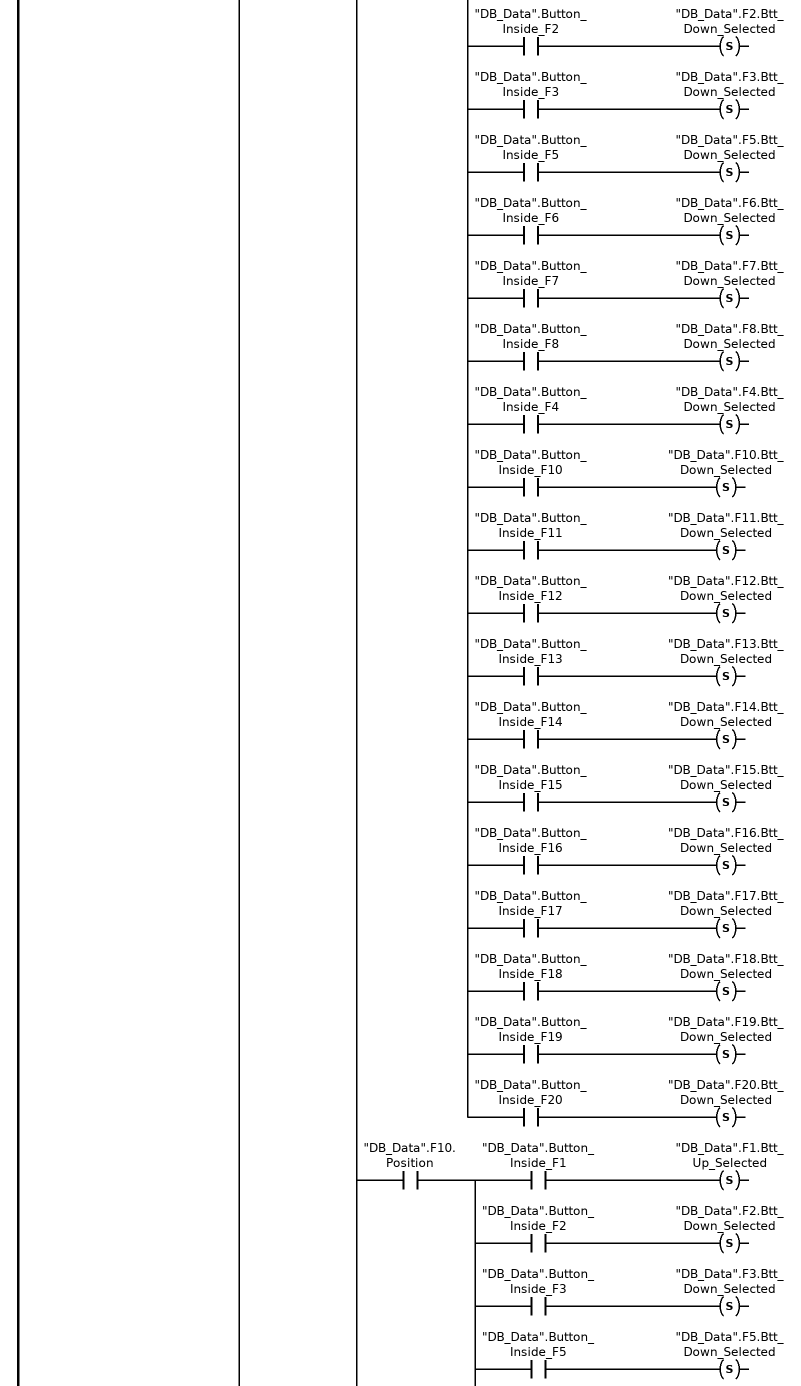
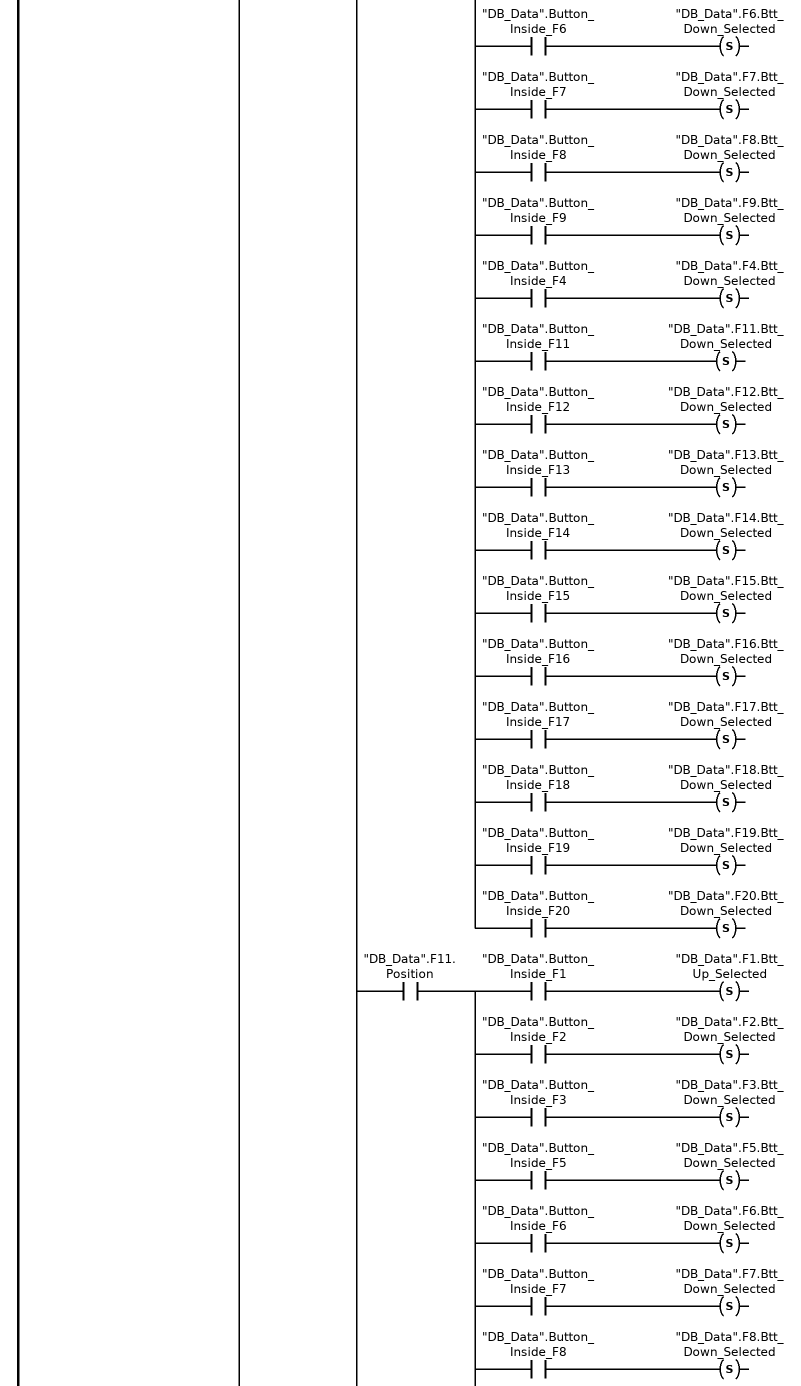
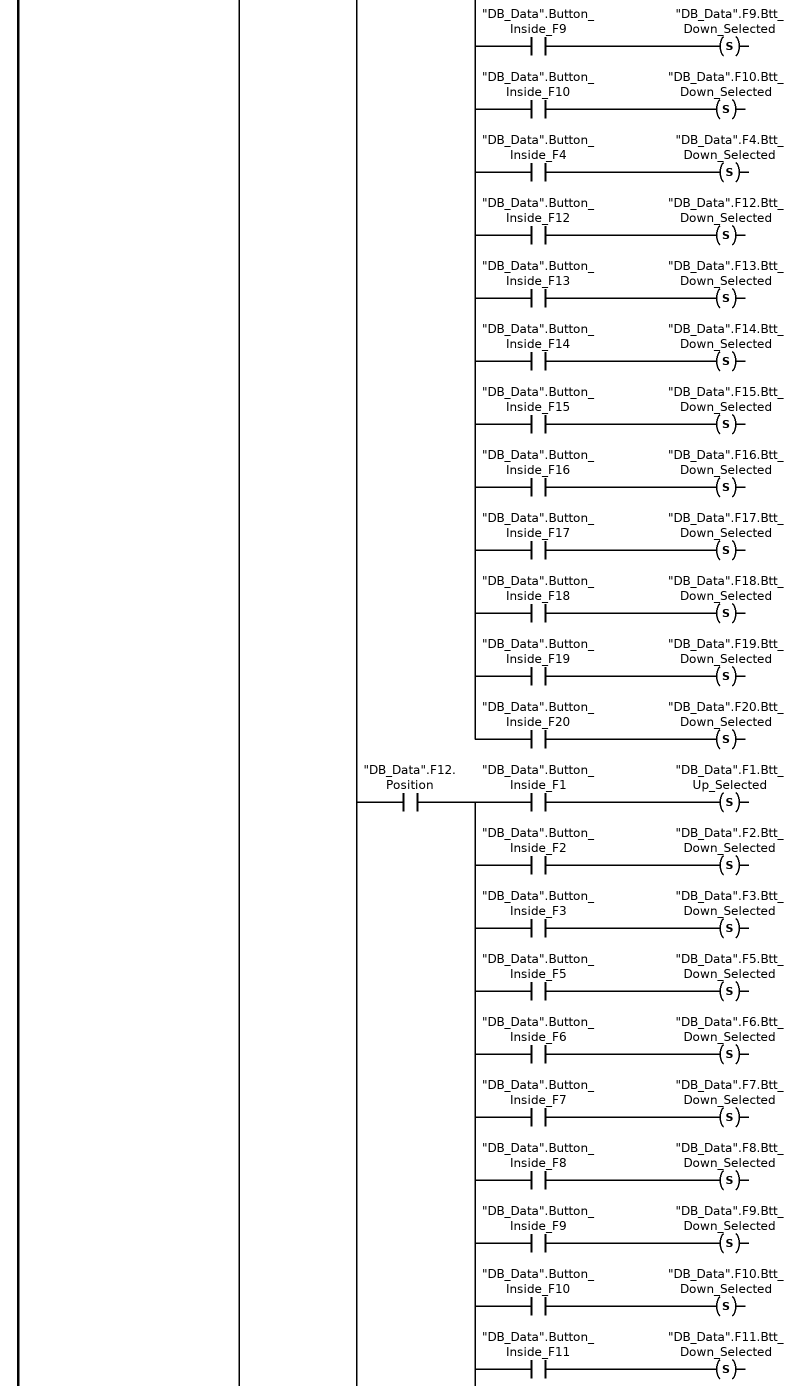
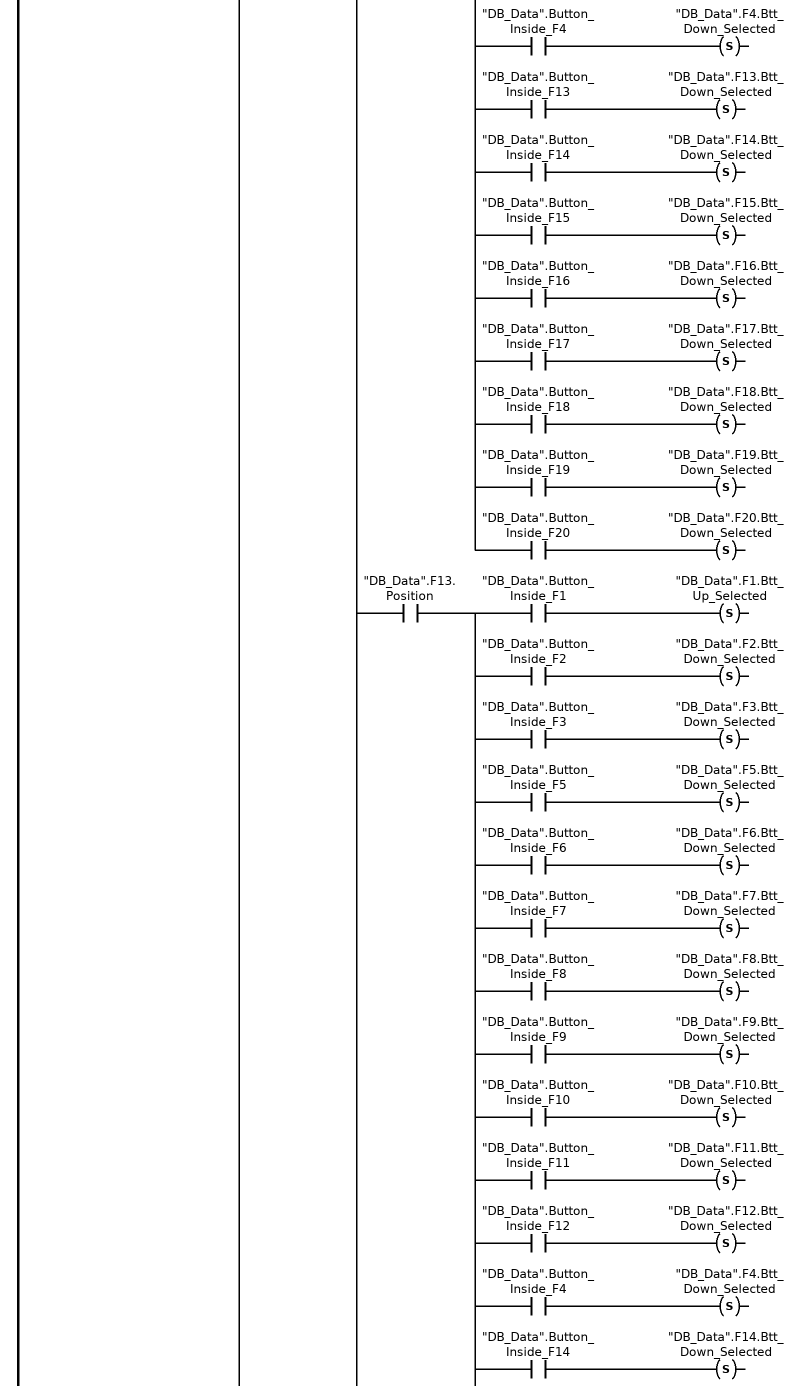
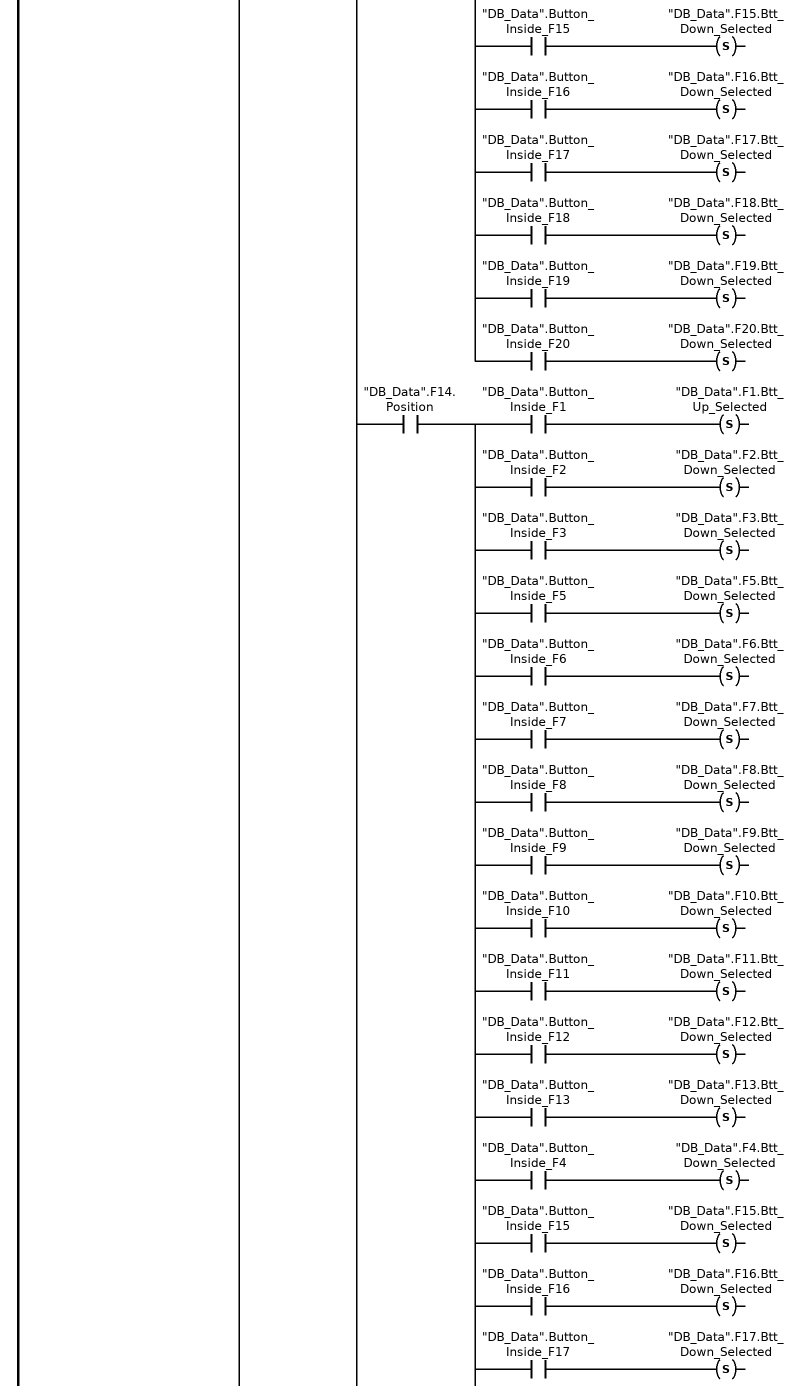
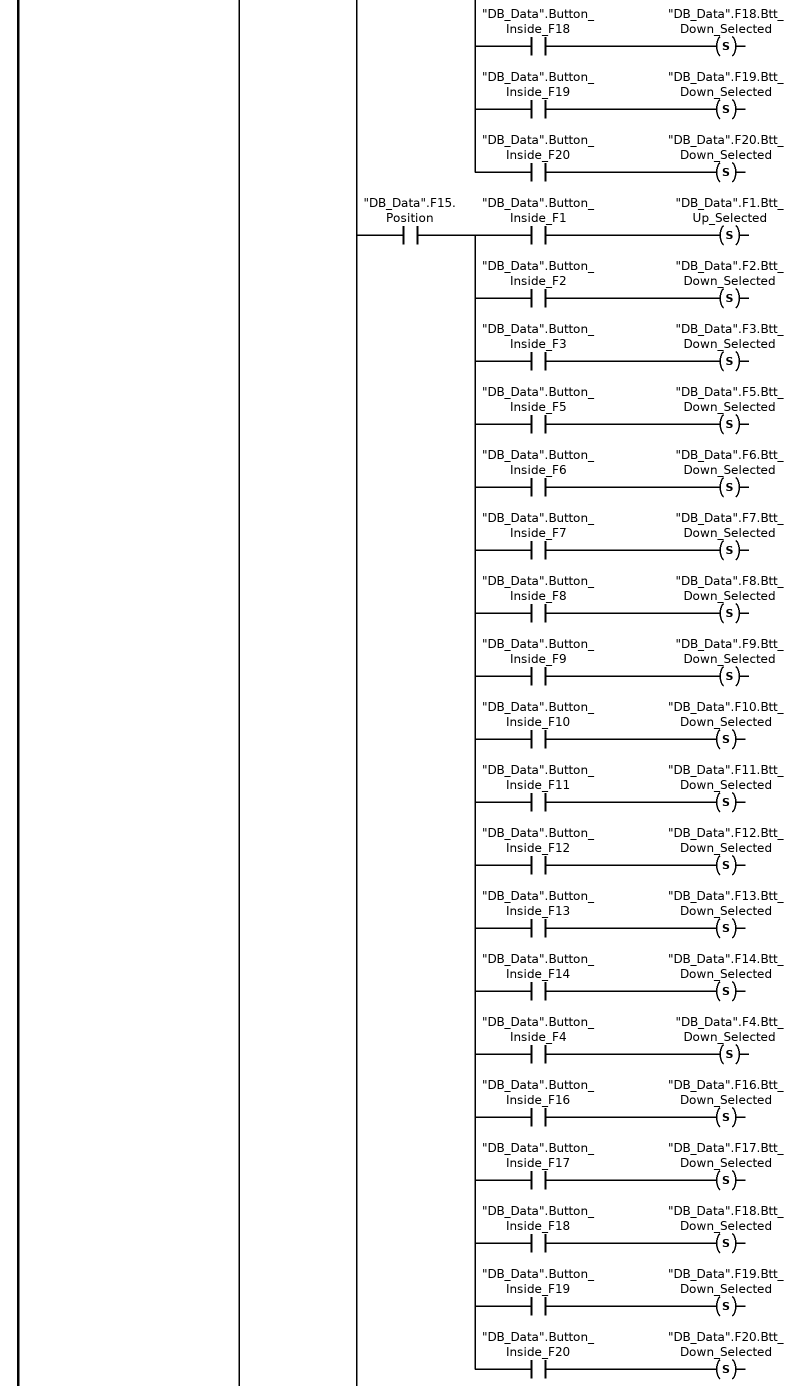
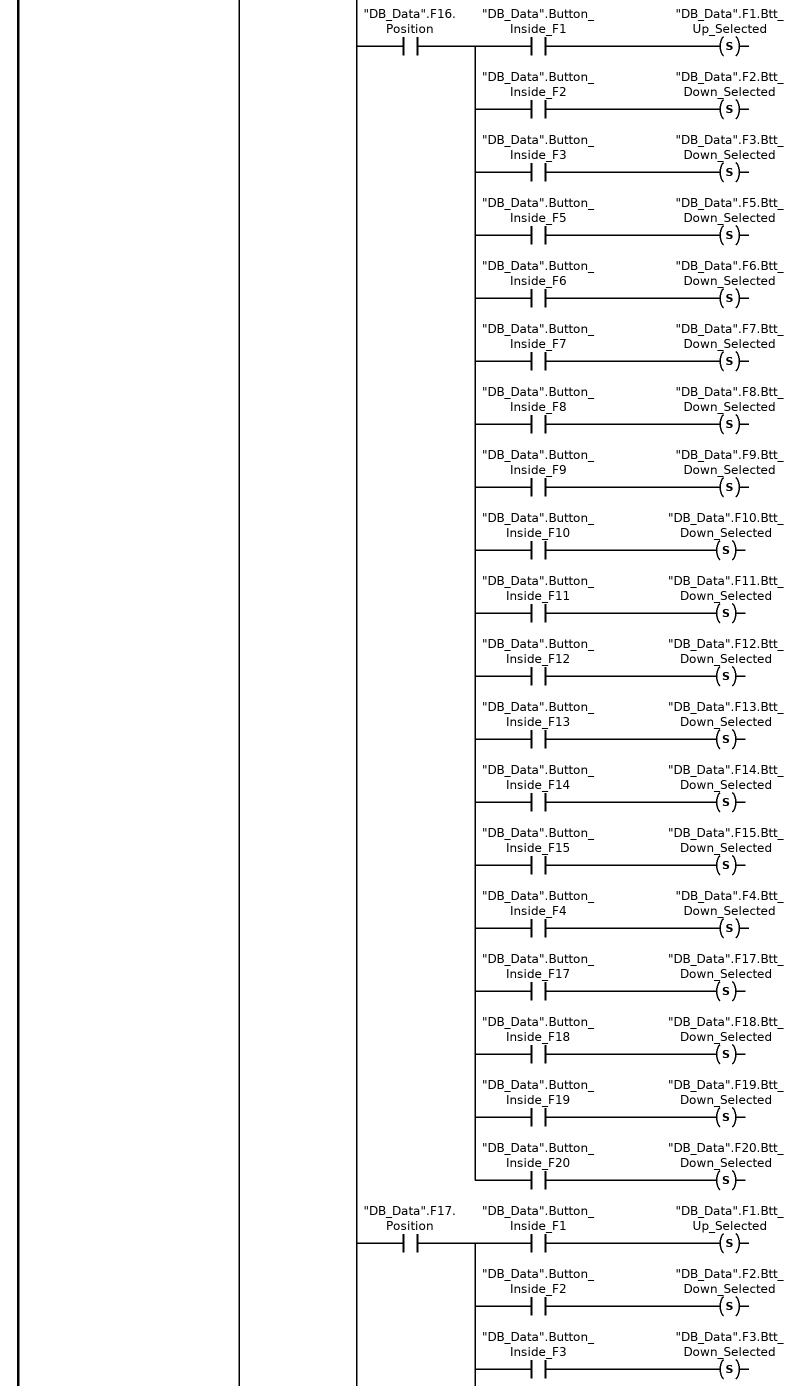
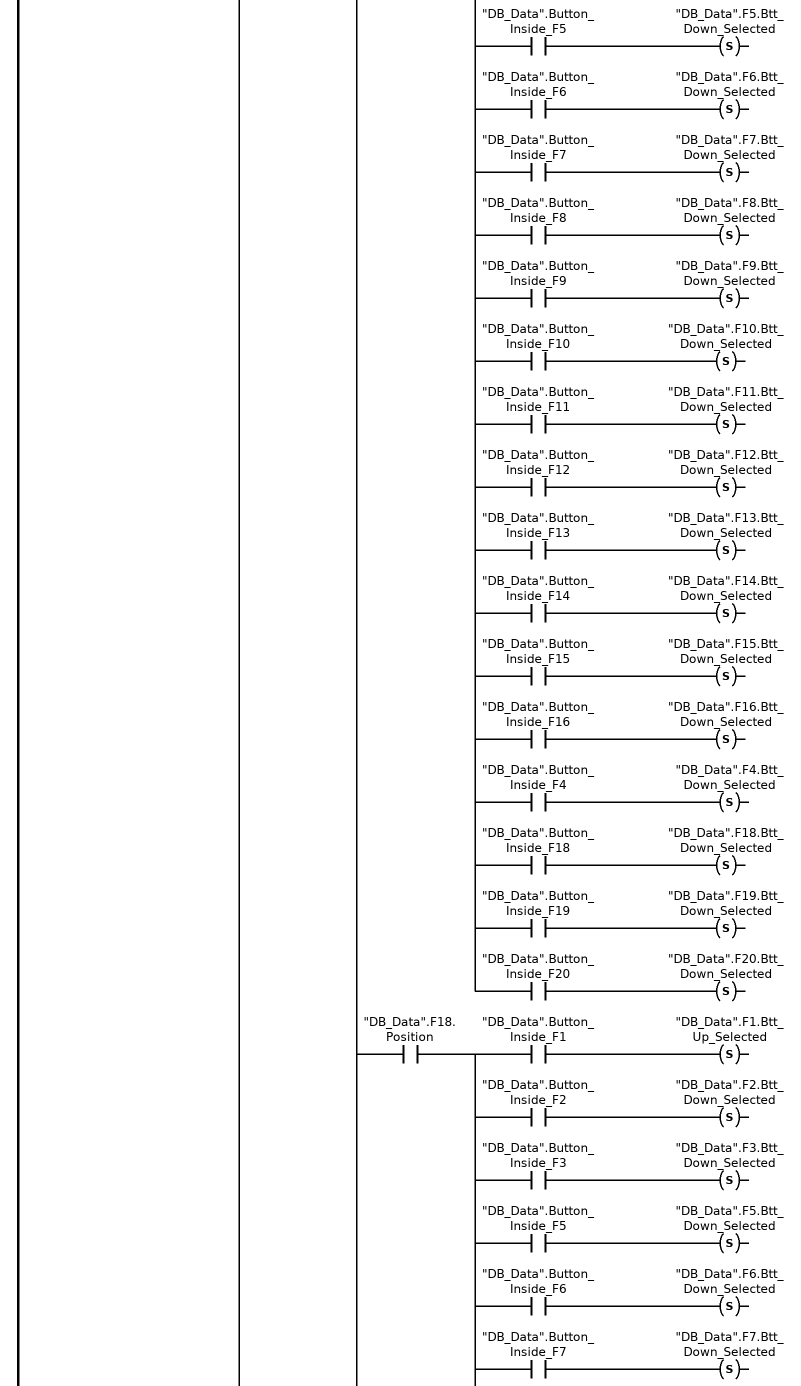
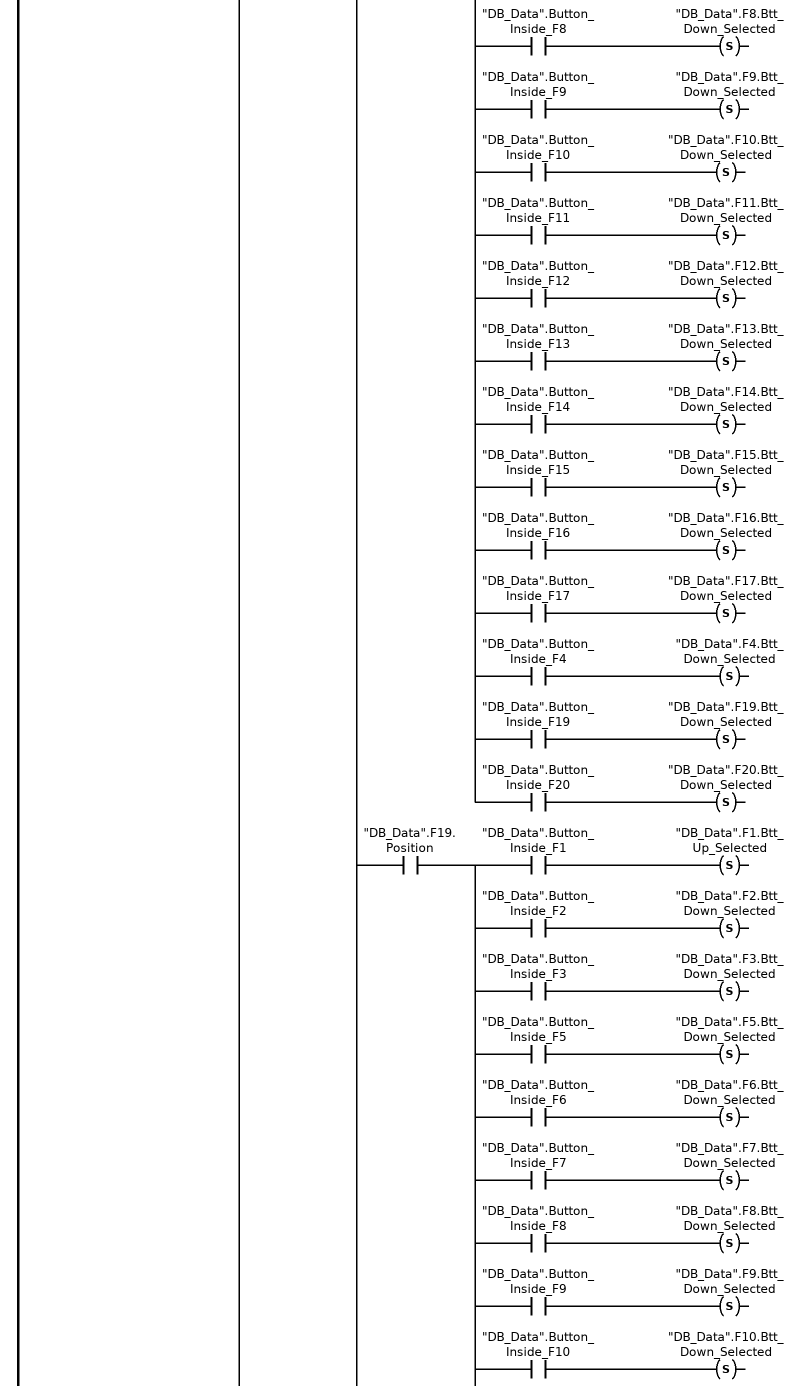
